LIN {X 0,Y 418.237,Z 526.484,A -85,B 0,C 180,E1 -10180.896,E2 -10180.896} C_VEL
LIN {X 0,Y 419.028,Z 517.254,A -85,B 0,C 180,E1 -10182.347,E2 -10182.347} C_VEL
LIN {X 0,Y 419.709,Z 507.688,A -85,B 0,C 180,E1 -10183.557,E2 -10183.557} C_VEL
LIN {X 0,Y 420.529,Z 497.102,A -85,B 0,C 180,E1 -10184.641,E2 -10184.641} C_VEL
LIN {X 0,Y 421.367,Z 485.277,A -85,B 0,C 180,E1 -10185.601,E2 -10185.601} C_VEL
LIN {X 0,Y 422.297,Z 472.62,A -85,B 0,C 180,E1 -10186.372,E2 -10186.372} C_VEL
LIN {X 0,Y 422.924,Z 459.994,A -85,B 0,C 180,E1 -10186.937,E2 -10186.937} C_VEL
LIN {X 0,Y 423.479,Z 446.573,A -85,B 0,C 180,E1 -10187.318,E2 -10187.318} C_VEL
LIN {X 0,Y 424.411,Z 367.767,A -85,B 0,C 180,E1 -10188.682,E2 -10188.682} C_VEL
LIN {X 0,Y 421.017,Z 346.244,A -85,B 0,C 180,E1 -10189.244,E2 -10189.244} C_VEL
LIN {X 0,Y 419.876,Z 339.849,A -85,B 0,C 180,E1 -10189.436,E2 -10189.436} C_VEL
LIN {X 0,Y 421.122,Z 320.957,A -85,B 0,C 180,E1 -10193,E2 -10193} C_VEL
LIN {X 0,Y 421.806,Z 311.137,A -85,B 0,C 180,E1 -10194.879,E2 -10194.879} C_VEL
LIN {X 0,Y 420.145,Z 301.746,A -85,B 0,C 180,E1 -10196.849,E2 -10196.849} C_VEL
LIN {X 0,Y 418.293,Z 293.389,A -85,B 0,C 180,E1 -10198.701,E2 -10198.701} C_VEL
LIN {X 0,Y 418.243,Z 293.391,A -85,B 0,C 180,E1 -10202.528,E2 -10202.528} C_VEL
LIN {X 0,Y 418.256,Z 293.389,A -85,B 0,C 180,E1 -10204.841,E2 -10204.841} C_VEL
LIN {X 0,Y 418.242,Z 293.39,A -85,B 0,C 180,E1 -10208.442,E2 -10208.442} C_VEL
LIN {X 0,Y 418.219,Z 293.387,A -85,B 0,C 180,E1 -10210.947,E2 -10210.947} C_VEL
LIN {X 0,Y 418.207,Z 293.389,A -85,B 0,C 180,E1 -10213.729,E2 -10213.729} C_VEL
LIN {X 0,Y 418.206,Z 293.391,A -85,B 0,C 180,E1 -10216.448,E2 -10216.448} C_VEL
LIN {X 0,Y 418.221,Z 293.385,A -85,B 0,C 180,E1 -10219.13,E2 -10219.13} C_VEL
LIN {X 0,Y 418.226,Z 293.386,A -85,B 0,C 180,E1 -10222.166,E2 -10222.166} C_VEL
LIN {X 0,Y 418.26,Z 293.378,A -85,B 0,C 180,E1 -10225.42,E2 -10225.42} C_VEL
LIN {X 0,Y 418.208,Z 293.388,A -85,B 0,C 180,E1 -10228.604,E2 -10228.604} C_VEL
LIN {X 0,Y 418.287,Z 293.375,A -85,B 0,C 180,E1 -10231.936,E2 -10231.936} C_VEL
LIN {X 0,Y 418.286,Z 293.375,A -85,B 0,C 180,E1 -10235.163,E2 -10235.163} C_VEL
LIN {X 0,Y 418.231,Z 293.387,A -85,B 0,C 180,E1 -10238.304,E2 -10238.304} C_VEL
LIN {X 0,Y 418.281,Z 293.38,A -85,B 0,C 180,E1 -10241.383,E2 -10241.383} C_VEL
LIN {X 0,Y 418.299,Z 293.375,A -85,B 0,C 180,E1 -10244.406,E2 -10244.406} C_VEL
LIN {X 0,Y 418.352,Z 293.366,A -85,B 0,C 180,E1 -10247.386,E2 -10247.386} C_VEL
LIN {X 0,Y 418.338,Z 293.374,A -85,B 0,C 180,E1 -10250.329,E2 -10250.329} C_VEL
LIN {X 0,Y 418.509,Z 293.347,A -85,B 0,C 180,E1 -10252.28,E2 -10252.28} C_VEL
LIN {X 0,Y 418.51,Z 293.351,A -85,B 0,C 180,E1 -10254.217,E2 -10254.217} C_VEL
LIN {X 0,Y 418.542,Z 293.346,A -85,B 0,C 180,E1 -10258.076,E2 -10258.076} C_VEL
LIN {X 0,Y 418.67,Z 293.327,A -85,B 0,C 180,E1 -10260,E2 -10260} C_VEL
LIN {X 0,Y 418.507,Z 293.356,A -85,B 0,C 180,E1 -10262.888,E2 -10262.888} C_VEL
LIN {X 0,Y 418.491,Z 293.355,A -85,B 0,C 180,E1 -10266.751,E2 -10266.751} C_VEL
LIN {X 0,Y 418.397,Z 293.366,A -85,B 0,C 180,E1 -10268.695,E2 -10268.695} C_VEL
LIN {X 0,Y 418.313,Z 293.375,A -85,B 0,C 180,E1 -10271.631,E2 -10271.631} C_VEL
LIN {X 0,Y 418.3,Z 293.376,A -85,B 0,C 180,E1 -10274.597,E2 -10274.597} C_VEL
LIN {X 0,Y 418.283,Z 293.378,A -85,B 0,C 180,E1 -10277.604,E2 -10277.604} C_VEL
LIN {X 0,Y 418.247,Z 293.385,A -85,B 0,C 180,E1 -10280.664,E2 -10280.664} C_VEL
LIN {X 0,Y 418.283,Z 293.379,A -85,B 0,C 180,E1 -10283.782,E2 -10283.782} C_VEL
LIN {X 0,Y 418.308,Z 293.38,A -85,B 0,C 180,E1 -10287.071,E2 -10287.071} C_VEL
LIN {X 0,Y 418.242,Z 293.383,A -85,B 0,C 180,E1 -10290.273,E2 -10290.273} C_VEL
LIN {X 0,Y 418.246,Z 293.385,A -85,B 0,C 180,E1 -10293.678,E2 -10293.678} C_VEL
LIN {X 0,Y 418.237,Z 293.389,A -85,B 0,C 180,E1 -10297.225,E2 -10297.225} C_VEL
LIN {X 0,Y 418.227,Z 293.388,A -85,B 0,C 180,E1 -10299.685,E2 -10299.685} C_VEL
LIN {X 0,Y 418.213,Z 293.388,A -85,B 0,C 180,E1 -10302.32,E2 -10302.32} C_VEL
LIN {X 0,Y 418.235,Z 293.39,A -85,B 0,C 180,E1 -10305.109,E2 -10305.109} C_VEL
LIN {X 0,Y 418.222,Z 293.39,A -85,B 0,C 180,E1 -10307.765,E2 -10307.765} C_VEL
LIN {X 0,Y 418.235,Z 293.39,A -85,B 0,C 180,E1 -10311.557,E2 -10311.557} C_VEL
LIN {X 0,Y 418.258,Z 293.381,A -85,B 0,C 180,E1 -10315.16,E2 -10315.16} C_VEL
LIN {X 0,Y 418.246,Z 293.386,A -85,B 0,C 180,E1 -10317.473,E2 -10317.473} C_VEL
LIN {X 0,Y 418.265,Z 293.452,A -85,B 0,C 180,E1 -10319.201,E2 -10319.201} C_VEL
LIN {X 0,Y 420.275,Z 303.434,A -85,B 0,C 180,E1 -10321.525,E2 -10321.525} C_VEL
LIN {X 0,Y 420.363,Z 304.121,A -85,B 0,C 180,E1 -10321.647,E2 -10321.647} C_VEL
LIN {X 0,Y 424.619,Z 321.891,A -85,B 0,C 180,E1 -10322.199,E2 -10322.199} C_VEL
LIN {X 0,Y 424.878,Z 325.308,A -85,B 0,C 180,E1 -10322.274,E2 -10322.274} C_VEL
LIN {X 0,Y 423.654,Z 411.995,A -85,B 0,C 180,E1 -10323.783,E2 -10323.783} C_VEL
LIN {X 0,Y 423.327,Z 425.918,A -85,B 0,C 180,E1 -10324.246,E2 -10324.246} C_VEL
LIN {X 0,Y 422.698,Z 438.277,A -85,B 0,C 180,E1 -10324.849,E2 -10324.849} C_VEL
LIN {X 0,Y 422.001,Z 450.37,A -85,B 0,C 180,E1 -10325.658,E2 -10325.658} C_VEL
LIN {X 0,Y 421.34,Z 460.803,A -85,B 0,C 180,E1 -10326.551,E2 -10326.551} C_VEL
LIN {X 0,Y 420.519,Z 471.216,A -85,B 0,C 180,E1 -10327.654,E2 -10327.654} C_VEL
LIN {X 0,Y 419.787,Z 480.656,A -85,B 0,C 180,E1 -10328.904,E2 -10328.904} C_VEL
LIN {X 0,Y 418.974,Z 489.748,A -85,B 0,C 180,E1 -10330.399,E2 -10330.399} C_VEL
LIN {X 0,Y 418.366,Z 497.004,A -85,B 0,C 180,E1 -10331.895,E2 -10331.895} C_VEL
LIN {X 0,Y 417.912,Z 502.928,A -85,B 0,C 180,E1 -10333.451,E2 -10333.451} C_VEL
LIN {X 0,Y 417.571,Z 507.193,A -85,B 0,C 180,E1 -10334.879,E2 -10334.879} C_VEL
LIN {X 0,Y 417.319,Z 510.544,A -85,B 0,C 180,E1 -10336.364,E2 -10336.364} C_VEL
LIN {X 0,Y 417.186,Z 512.718,A -85,B 0,C 180,E1 -10337.712,E2 -10337.712} C_VEL
LIN {X 0,Y 417.034,Z 514.334,A -85,B 0,C 180,E1 -10339.52,E2 -10339.52} C_VEL
LIN {X 0,Y 417.041,Z 514.637,A -85,B 0,C 180,E1 -10341.277,E2 -10341.277} C_VEL
LIN {X 0,Y 417.072,Z 514.25,A -85,B 0,C 180,E1 -10342.253,E2 -10342.253} C_VEL
LIN {X 0,Y 417.181,Z 512.868,A -85,B 0,C 180,E1 -10343.724,E2 -10343.724} C_VEL
LIN {X 0,Y 416.533,Z 511.788,A -85,B 0,C 180,E1 -10344.516,E2 -10344.516} C_VEL
LIN {X 0,Y 413.788,Z 509.541,A -85,B 0,C 180,E1 -10345.795,E2 -10345.795} C_VEL
LIN {X 0,Y 411.494,Z 507.287,A -85,B 0,C 180,E1 -10346.808,E2 -10346.808} C_VEL
LIN {X 0,Y 410.54,Z 505.221,A -85,B 0,C 180,E1 -10347.572,E2 -10347.572} C_VEL
LIN {X 0,Y 410.478,Z 504.425,A -85,B 0,C 180,E1 -10347.826,E2 -10347.826} C_VEL
LIN {X 0,Y 410.657,Z 500.332,A -85,B 0,C 180,E1 -10349.02,E2 -10349.02} C_VEL
LIN {X 0,Y 411.218,Z 494.07,A -85,B 0,C 180,E1 -10350.49,E2 -10350.49} C_VEL
LIN {X 0,Y 411.727,Z 486.262,A -85,B 0,C 180,E1 -10351.957,E2 -10351.957} C_VEL
LIN {X 0,Y 412.392,Z 476.551,A -85,B 0,C 180,E1 -10353.42,E2 -10353.42} C_VEL
LIN {X 0,Y 413.042,Z 466.441,A -85,B 0,C 180,E1 -10354.636,E2 -10354.636} C_VEL
LIN {X 0,Y 413.78,Z 455.013,A -85,B 0,C 180,E1 -10355.727,E2 -10355.727} C_VEL
LIN {X 0,Y 414.492,Z 443.752,A -85,B 0,C 180,E1 -10356.573,E2 -10356.573} C_VEL
LIN {X 0,Y 414.845,Z 432.31,A -85,B 0,C 180,E1 -10357.239,E2 -10357.239} C_VEL
LIN {X 0,Y 415.282,Z 419.113,A -85,B 0,C 180,E1 -10357.782,E2 -10357.782} C_VEL
LIN {X 0,Y 415.62,Z 406.202,A -85,B 0,C 180,E1 -10358.112,E2 -10358.112} C_VEL
LIN {X 0,Y 416.569,Z 323.375,A -85,B 0,C 180,E1 -10359.537,E2 -10359.537} C_VEL
LIN {X 0,Y 412.825,Z 304.032,A -85,B 0,C 180,E1 -10360.041,E2 -10360.041} C_VEL
LIN {X 0,Y 411.358,Z 294.341,A -85,B 0,C 180,E1 -10362.238,E2 -10362.238} C_VEL
LIN {X 0,Y 411.258,Z 294.253,A -85,B 0,C 180,E1 -10365.869,E2 -10365.869} C_VEL
LIN {X 0,Y 411.224,Z 294.262,A -85,B 0,C 180,E1 -10368.949,E2 -10368.949} C_VEL
LIN {X 0,Y 411.205,Z 294.264,A -85,B 0,C 180,E1 -10372.641,E2 -10372.641} C_VEL
LIN {X 0,Y 411.189,Z 294.264,A -85,B 0,C 180,E1 -10375.297,E2 -10375.297} C_VEL
LIN {X 0,Y 411.177,Z 294.266,A -85,B 0,C 180,E1 -10378.594,E2 -10378.594} C_VEL
LIN {X 0,Y 411.168,Z 294.263,A -85,B 0,C 180,E1 -10381.998,E2 -10381.998} C_VEL
LIN {X 0,Y 411.208,Z 294.264,A -85,B 0,C 180,E1 -10384.877,E2 -10384.877} C_VEL
LIN {X 0,Y 411.2,Z 294.259,A -85,B 0,C 180,E1 -10388.167,E2 -10388.167} C_VEL
LIN {X 0,Y 411.165,Z 294.265,A -85,B 0,C 180,E1 -10391.808,E2 -10391.808} C_VEL
LIN {X 0,Y 411.179,Z 294.267,A -85,B 0,C 180,E1 -10395.509,E2 -10395.509} C_VEL
LIN {X 0,Y 411.152,Z 294.267,A -85,B 0,C 180,E1 -10398.775,E2 -10398.775} C_VEL
LIN {X 0,Y 411.188,Z 294.263,A -85,B 0,C 180,E1 -10402.025,E2 -10402.025} C_VEL
LIN {X 0,Y 411.207,Z 294.261,A -85,B 0,C 180,E1 -10405.123,E2 -10405.123} C_VEL
LIN {X 0,Y 411.169,Z 294.266,A -85,B 0,C 180,E1 -10408.003,E2 -10408.003} C_VEL
LIN {X 0,Y 411.198,Z 294.264,A -85,B 0,C 180,E1 -10411.408,E2 -10411.408} C_VEL
LIN {X 0,Y 411.217,Z 294.258,A -85,B 0,C 180,E1 -10414.934,E2 -10414.934} C_VEL
LIN {X 0,Y 411.208,Z 294.265,A -85,B 0,C 180,E1 -10417.913,E2 -10417.913} C_VEL
LIN {X 0,Y 411.223,Z 294.257,A -85,B 0,C 180,E1 -10421.051,E2 -10421.051} C_VEL
LIN {X 0,Y 411.258,Z 294.258,A -85,B 0,C 180,E1 -10424.131,E2 -10424.131} C_VEL
LIN {X 0,Y 411.307,Z 294.246,A -85,B 0,C 180,E1 -10427.165,E2 -10427.165} C_VEL
LIN {X 0,Y 411.282,Z 294.256,A -85,B 0,C 180,E1 -10430.161,E2 -10430.161} C_VEL
LIN {X 0,Y 411.395,Z 294.235,A -85,B 0,C 180,E1 -10433.132,E2 -10433.132} C_VEL
LIN {X 0,Y 411.293,Z 294.248,A -85,B 0,C 180,E1 -10435.099,E2 -10435.099} C_VEL
LIN {X 0,Y 411.506,Z 294.226,A -85,B 0,C 180,E1 -10438.042,E2 -10438.042} C_VEL
LIN {X 0,Y 411.421,Z 294.233,A -85,B 0,C 180,E1 -10440.979,E2 -10440.979} C_VEL
LIN {X 0,Y 411.43,Z 294.232,A -85,B 0,C 180,E1 -10442.937,E2 -10442.937} C_VEL
LIN {X 0,Y 411.394,Z 294.238,A -85,B 0,C 180,E1 -10446.868,E2 -10446.868} C_VEL
LIN {X 0,Y 411.278,Z 294.251,A -85,B 0,C 180,E1 -10449.839,E2 -10449.839} C_VEL
LIN {X 0,Y 411.309,Z 294.248,A -85,B 0,C 180,E1 -10453.103,E2 -10453.103} C_VEL
LIN {X 0,Y 411.261,Z 294.257,A -85,B 0,C 180,E1 -10456.888,E2 -10456.888} C_VEL
LIN {X 0,Y 411.235,Z 294.256,A -85,B 0,C 180,E1 -10459.986,E2 -10459.986} C_VEL
LIN {X 0,Y 411.191,Z 294.264,A -85,B 0,C 180,E1 -10463.148,E2 -10463.148} C_VEL
LIN {X 0,Y 411.178,Z 294.264,A -85,B 0,C 180,E1 -10466.385,E2 -10466.385} C_VEL
LIN {X 0,Y 411.198,Z 294.26,A -85,B 0,C 180,E1 -10469.713,E2 -10469.713} C_VEL
LIN {X 0,Y 411.207,Z 294.265,A -85,B 0,C 180,E1 -10473.156,E2 -10473.156} C_VEL
LIN {X 0,Y 411.195,Z 294.262,A -85,B 0,C 180,E1 -10476.552,E2 -10476.552} C_VEL
LIN {X 0,Y 411.172,Z 294.264,A -85,B 0,C 180,E1 -10479.72,E2 -10479.72} C_VEL
LIN {X 0,Y 411.165,Z 294.27,A -85,B 0,C 180,E1 -10483.135,E2 -10483.135} C_VEL
LIN {X 0,Y 411.166,Z 294.265,A -85,B 0,C 180,E1 -10485.881,E2 -10485.881} C_VEL
LIN {X 0,Y 411.16,Z 294.271,A -85,B 0,C 180,E1 -10489.492,E2 -10489.492} C_VEL
LIN {X 0,Y 411.185,Z 294.263,A -85,B 0,C 180,E1 -10492.025,E2 -10492.025} C_VEL
LIN {X 0,Y 411.205,Z 294.262,A -85,B 0,C 180,E1 -10495.123,E2 -10495.123} C_VEL
LIN {X 0,Y 411.167,Z 294.27,A -85,B 0,C 180,E1 -10498.002,E2 -10498.002} C_VEL
LIN {X 0,Y 411.214,Z 294.264,A -85,B 0,C 180,E1 -10501.409,E2 -10501.409} C_VEL
LIN {X 0,Y 411.262,Z 294.307,A -85,B 0,C 180,E1 -10502.073,E2 -10502.073} C_VEL
LIN {X 0,Y 413.901,Z 307.893,A -85,B 0,C 180,E1 -10504.88,E2 -10504.88} C_VEL
LIN {X 0,Y 414.052,Z 312.05,A -85,B 0,C 180,E1 -10505.693,E2 -10505.693} C_VEL
LIN {X 0,Y 412.954,Z 329.844,A -85,B 0,C 180,E1 -10509.059,E2 -10509.059} C_VEL
LIN {X 0,Y 412.351,Z 339.884,A -85,B 0,C 180,E1 -10510.943,E2 -10510.943} C_VEL
LIN {X 0,Y 416.255,Z 368.768,A -85,B 0,C 180,E1 -10511.625,E2 -10511.625} C_VEL
LIN {X 0,Y 415.383,Z 449.072,A -85,B 0,C 180,E1 -10513.03,E2 -10513.03} C_VEL
LIN {X 0,Y 414.775,Z 463.016,A -85,B 0,C 180,E1 -10513.48,E2 -10513.48} C_VEL
LIN {X 0,Y 414.176,Z 476.032,A -85,B 0,C 180,E1 -10514.12,E2 -10514.12} C_VEL
LIN {X 0,Y 413.358,Z 488.654,A -85,B 0,C 180,E1 -10514.972,E2 -10514.972} C_VEL
LIN {X 0,Y 412.697,Z 500.406,A -85,B 0,C 180,E1 -10516.003,E2 -10516.003} C_VEL
LIN {X 0,Y 411.956,Z 511.029,A -85,B 0,C 180,E1 -10517.186,E2 -10517.186} C_VEL
LIN {X 0,Y 411.342,Z 520.018,A -85,B 0,C 180,E1 -10518.418,E2 -10518.418} C_VEL
LIN {X 0,Y 410.749,Z 528.786,A -85,B 0,C 180,E1 -10519.899,E2 -10519.899} C_VEL
LIN {X 0,Y 410.387,Z 535.776,A -85,B 0,C 180,E1 -10521.381,E2 -10521.381} C_VEL
LIN {X 0,Y 410.162,Z 542.192,A -85,B 0,C 180,E1 -10523.111,E2 -10523.111} C_VEL
LIN {X 0,Y 410.032,Z 546.387,A -85,B 0,C 180,E1 -10524.59,E2 -10524.59} C_VEL
LIN {X 0,Y 409.943,Z 549.506,A -85,B 0,C 180,E1 -10526.067,E2 -10526.067} C_VEL
LIN {X 0,Y 409.987,Z 551.061,A -85,B 0,C 180,E1 -10527.052,E2 -10527.052} C_VEL
LIN {X 0,Y 410.019,Z 552.161,A -85,B 0,C 180,E1 -10528.035,E2 -10528.035} C_VEL
LIN {X 0,Y 409.973,Z 553.147,A -85,B 0,C 180,E1 -10529.999,E2 -10529.999} C_VEL
LIN {X 0,Y 409.978,Z 553.06,A -85,B 0,C 180,E1 -10530.982,E2 -10530.982} C_VEL
LIN {X 0,Y 410.018,Z 552.548,A -85,B 0,C 180,E1 -10531.964,E2 -10531.964} C_VEL
LIN {X 0,Y 409.969,Z 551.622,A -85,B 0,C 180,E1 -10532.947,E2 -10532.947} C_VEL
LIN {X 0,Y 410.02,Z 548.582,A -85,B 0,C 180,E1 -10534.916,E2 -10534.916} C_VEL
LIN {X 0,Y 410.041,Z 545.565,A -85,B 0,C 180,E1 -10536.223,E2 -10536.223} C_VEL
LIN {X 0,Y 410.283,Z 540.602,A -85,B 0,C 180,E1 -10537.876,E2 -10537.876} C_VEL
LIN {X 0,Y 410.702,Z 533.771,A -85,B 0,C 180,E1 -10539.604,E2 -10539.604} C_VEL
LIN {X 0,Y 411.253,Z 526.369,A -85,B 0,C 180,E1 -10541.084,E2 -10541.084} C_VEL
LIN {X 0,Y 412.072,Z 517.205,A -85,B 0,C 180,E1 -10542.559,E2 -10542.559} C_VEL
LIN {X 0,Y 412.81,Z 507.705,A -85,B 0,C 180,E1 -10543.788,E2 -10543.788} C_VEL
LIN {X 0,Y 413.65,Z 497.196,A -85,B 0,C 180,E1 -10544.89,E2 -10544.89} C_VEL
LIN {X 0,Y 414.555,Z 485.515,A -85,B 0,C 180,E1 -10545.864,E2 -10545.864} C_VEL
LIN {X 0,Y 415.517,Z 473.045,A -85,B 0,C 180,E1 -10546.647,E2 -10546.647} C_VEL
LIN {X 0,Y 416.215,Z 459.929,A -85,B 0,C 180,E1 -10547.25,E2 -10547.25} C_VEL
LIN {X 0,Y 416.778,Z 446.777,A -85,B 0,C 180,E1 -10547.637,E2 -10547.637} C_VEL
LIN {X 0,Y 417.744,Z 368.102,A -85,B 0,C 180,E1 -10549.023,E2 -10549.023} C_VEL
LIN {X 0,Y 414.43,Z 347.438,A -85,B 0,C 180,E1 -10549.58,E2 -10549.58} C_VEL
LIN {X 0,Y 413.028,Z 339.466,A -85,B 0,C 180,E1 -10549.826,E2 -10549.826} C_VEL
LIN {X 0,Y 414.155,Z 323.075,A -85,B 0,C 180,E1 -10552.972,E2 -10552.972} C_VEL
LIN {X 0,Y 414.904,Z 312.386,A -85,B 0,C 180,E1 -10555.053,E2 -10555.053} C_VEL
LIN {X 0,Y 413.209,Z 303.005,A -85,B 0,C 180,E1 -10557.063,E2 -10557.063} C_VEL
LIN {X 0,Y 411.224,Z 294.269,A -85,B 0,C 180,E1 -10559.041,E2 -10559.041} C_VEL
LIN {X 0,Y 411.163,Z 294.27,A -85,B 0,C 180,E1 -10561.997,E2 -10561.997} C_VEL
LIN {X 0,Y 411.207,Z 294.267,A -85,B 0,C 180,E1 -10564.878,E2 -10564.878} C_VEL
LIN {X 0,Y 411.196,Z 294.267,A -85,B 0,C 180,E1 -10568.167,E2 -10568.167} C_VEL
LIN {X 0,Y 411.161,Z 294.265,A -85,B 0,C 180,E1 -10571.228,E2 -10571.228} C_VEL
LIN {X 0,Y 411.173,Z 294.27,A -85,B 0,C 180,E1 -10574.49,E2 -10574.49} C_VEL
LIN {X 0,Y 411.175,Z 294.268,A -85,B 0,C 180,E1 -10578.194,E2 -10578.194} C_VEL
LIN {X 0,Y 411.219,Z 294.261,A -85,B 0,C 180,E1 -10580.776,E2 -10580.776} C_VEL
LIN {X 0,Y 411.194,Z 294.264,A -85,B 0,C 180,E1 -10584.471,E2 -10584.471} C_VEL
LIN {X 0,Y 411.203,Z 294.262,A -85,B 0,C 180,E1 -10586.873,E2 -10586.873} C_VEL
LIN {X 0,Y 411.229,Z 294.261,A -85,B 0,C 180,E1 -10590.644,E2 -10590.644} C_VEL
LIN {X 0,Y 411.233,Z 294.255,A -85,B 0,C 180,E1 -10593.619,E2 -10593.619} C_VEL
LIN {X 0,Y 411.198,Z 294.265,A -85,B 0,C 180,E1 -10596.852,E2 -10596.852} C_VEL
LIN {X 0,Y 411.211,Z 294.254,A -85,B 0,C 180,E1 -10600.05,E2 -10600.05} C_VEL
LIN {X 0,Y 411.259,Z 294.251,A -85,B 0,C 180,E1 -10603.131,E2 -10603.131} C_VEL
LIN {X 0,Y 411.302,Z 294.249,A -85,B 0,C 180,E1 -10606.896,E2 -10606.896} C_VEL
LIN {X 0,Y 411.29,Z 294.251,A -85,B 0,C 180,E1 -10610.161,E2 -10610.161} C_VEL
LIN {X 0,Y 411.478,Z 294.222,A -85,B 0,C 180,E1 -10612.147,E2 -10612.147} C_VEL
LIN {X 0,Y 411.472,Z 294.227,A -85,B 0,C 180,E1 -10614.118,E2 -10614.118} C_VEL
LIN {X 0,Y 411.511,Z 294.221,A -85,B 0,C 180,E1 -10618.043,E2 -10618.043} C_VEL
LIN {X 0,Y 411.639,Z 294.203,A -85,B 0,C 180,E1 -10620,E2 -10620} C_VEL
LIN {X 0,Y 411.462,Z 294.234,A -85,B 0,C 180,E1 -10622.937,E2 -10622.937} C_VEL
LIN {X 0,Y 411.458,Z 294.232,A -85,B 0,C 180,E1 -10626.867,E2 -10626.867} C_VEL
LIN {X 0,Y 411.29,Z 294.247,A -85,B 0,C 180,E1 -10629.839,E2 -10629.839} C_VEL
LIN {X 0,Y 411.302,Z 294.248,A -85,B 0,C 180,E1 -10633.105,E2 -10633.105} C_VEL
LIN {X 0,Y 411.254,Z 294.257,A -85,B 0,C 180,E1 -10636.889,E2 -10636.889} C_VEL
LIN {X 0,Y 411.228,Z 294.257,A -85,B 0,C 180,E1 -10639.987,E2 -10639.987} C_VEL
LIN {X 0,Y 411.2,Z 294.267,A -85,B 0,C 180,E1 -10643.148,E2 -10643.148} C_VEL
LIN {X 0,Y 411.234,Z 294.256,A -85,B 0,C 180,E1 -10646.382,E2 -10646.382} C_VEL
LIN {X 0,Y 411.198,Z 294.263,A -85,B 0,C 180,E1 -10649.713,E2 -10649.713} C_VEL
LIN {X 0,Y 411.205,Z 294.261,A -85,B 0,C 180,E1 -10653.157,E2 -10653.157} C_VEL
LIN {X 0,Y 411.191,Z 294.261,A -85,B 0,C 180,E1 -10656.553,E2 -10656.553} C_VEL
LIN {X 0,Y 411.194,Z 294.264,A -85,B 0,C 180,E1 -10659.725,E2 -10659.725} C_VEL
LIN {X 0,Y 411.164,Z 294.269,A -85,B 0,C 180,E1 -10663.135,E2 -10663.135} C_VEL
LIN {X 0,Y 411.164,Z 294.269,A -85,B 0,C 180,E1 -10665.882,E2 -10665.882} C_VEL
LIN {X 0,Y 411.148,Z 294.27,A -85,B 0,C 180,E1 -10668.775,E2 -10668.775} C_VEL
LIN {X 0,Y 411.183,Z 294.266,A -85,B 0,C 180,E1 -10672.026,E2 -10672.026} C_VEL
LIN {X 0,Y 411.205,Z 294.265,A -85,B 0,C 180,E1 -10675.667,E2 -10675.667} C_VEL
LIN {X 0,Y 411.2,Z 294.319,A -85,B 0,C 180,E1 -10678.878,E2 -10678.878} C_VEL
LIN {X 0,Y 413.33,Z 304.267,A -85,B 0,C 180,E1 -10681.243,E2 -10681.243} C_VEL
LIN {X 0,Y 416.615,Z 316.53,A -85,B 0,C 180,E1 -10681.664,E2 -10681.664} C_VEL
LIN {X 0,Y 418.302,Z 325.142,A -85,B 0,C 180,E1 -10681.915,E2 -10681.915} C_VEL
LIN {X 0,Y 416.98,Z 411.971,A -85,B 0,C 180,E1 -10683.444,E2 -10683.444} C_VEL
LIN {X 0,Y 416.657,Z 425.074,A -85,B 0,C 180,E1 -10683.876,E2 -10683.876} C_VEL
LIN {X 0,Y 416.037,Z 437.678,A -85,B 0,C 180,E1 -10684.485,E2 -10684.485} C_VEL
LIN {X 0,Y 415.362,Z 449.209,A -85,B 0,C 180,E1 -10685.243,E2 -10685.243} C_VEL
LIN {X 0,Y 414.663,Z 459.822,A -85,B 0,C 180,E1 -10686.141,E2 -10686.141} C_VEL
LIN {X 0,Y 413.78,Z 470.539,A -85,B 0,C 180,E1 -10687.27,E2 -10687.27} C_VEL
LIN {X 0,Y 412.969,Z 480.214,A -85,B 0,C 180,E1 -10688.538,E2 -10688.538} C_VEL
LIN {X 0,Y 412.245,Z 487.972,A -85,B 0,C 180,E1 -10689.789,E2 -10689.789} C_VEL
LIN {X 0,Y 411.564,Z 495.689,A -85,B 0,C 180,E1 -10691.327,E2 -10691.327} C_VEL
LIN {X 0,Y 410.948,Z 502.674,A -85,B 0,C 180,E1 -10693.099,E2 -10693.099} C_VEL
LIN {X 0,Y 410.567,Z 507.232,A -85,B 0,C 180,E1 -10694.614,E2 -10694.614} C_VEL
LIN {X 0,Y 410.297,Z 510.665,A -85,B 0,C 180,E1 -10696.126,E2 -10696.126} C_VEL
LIN {X 0,Y 410.13,Z 513.062,A -85,B 0,C 180,E1 -10697.624,E2 -10697.624} C_VEL
LIN {X 0,Y 409.994,Z 514.513,A -85,B 0,C 180,E1 -10699.132,E2 -10699.132} C_VEL
LIN {X 0,Y 409.908,Z 514.954,A -85,B 0,C 180,E1 -10700.128,E2 -10700.128} C_VEL
LIN {X 0,Y 409.976,Z 514.638,A -85,B 0,C 180,E1 -10702.118,E2 -10702.118} C_VEL
LIN {X 0,Y 410.09,Z 513.202,A -85,B 0,C 180,E1 -10703.731,E2 -10703.731} C_VEL
LIN {X 0,Y 410.121,Z 511.149,A -85,B 0,C 180,E1 -10705.085,E2 -10705.085} C_VEL
LIN {X 0,Y 410.328,Z 507.976,A -85,B 0,C 180,E1 -10706.564,E2 -10706.564} C_VEL
LIN {X 0,Y 410.478,Z 504.425,A -85,B 0,C 180,E1 -10707.826,E2 -10707.826} C_VEL
LIN {X 0,Y 409.915,Z 502.016,A -85,B 0,C 180,E1 -10708.576,E2 -10708.576} C_VEL
LIN {X 0,Y 406.247,Z 495.799,A -85,B 0,C 180,E1 -10710.245,E2 -10710.245} C_VEL
LIN {X 0,Y 404.654,Z 491.638,A -85,B 0,C 180,E1 -10711.171,E2 -10711.171} C_VEL
LIN {X 0,Y 404.508,Z 489.298,A -85,B 0,C 180,E1 -10711.622,E2 -10711.622} C_VEL
LIN {X 0,Y 405.101,Z 481.13,A -85,B 0,C 180,E1 -10712.984,E2 -10712.984} C_VEL
LIN {X 0,Y 405.734,Z 472.036,A -85,B 0,C 180,E1 -10714.222,E2 -10714.222} C_VEL
LIN {X 0,Y 406.39,Z 461.925,A -85,B 0,C 180,E1 -10715.334,E2 -10715.334} C_VEL
LIN {X 0,Y 407.183,Z 450.692,A -85,B 0,C 180,E1 -10716.318,E2 -10716.318} C_VEL
LIN {X 0,Y 407.684,Z 440.078,A -85,B 0,C 180,E1 -10717.056,E2 -10717.056} C_VEL
LIN {X 0,Y 408.133,Z 428.554,A -85,B 0,C 180,E1 -10717.67,E2 -10717.67} C_VEL
LIN {X 0,Y 408.508,Z 416.317,A -85,B 0,C 180,E1 -10718.129,E2 -10718.129} C_VEL
LIN {X 0,Y 408.786,Z 400.812,A -85,B 0,C 180,E1 -10718.466,E2 -10718.466} C_VEL
LIN {X 0,Y 409.75,Z 324.356,A -85,B 0,C 180,E1 -10719.799,E2 -10719.799} C_VEL
LIN {X 0,Y 406.056,Z 305.517,A -85,B 0,C 180,E1 -10720.296,E2 -10720.296} C_VEL
LIN {X 0,Y 405.79,Z 304.263,A -85,B 0,C 180,E1 -10720.353,E2 -10720.353} C_VEL
LIN {X 0,Y 404.288,Z 295.127,A -85,B 0,C 180,E1 -10722.487,E2 -10722.487} C_VEL
LIN {X 0,Y 404.226,Z 295.13,A -85,B 0,C 180,E1 -10726.152,E2 -10726.152} C_VEL
LIN {X 0,Y 404.168,Z 295.137,A -85,B 0,C 180,E1 -10729.293,E2 -10729.293} C_VEL
LIN {X 0,Y 404.152,Z 295.145,A -85,B 0,C 180,E1 -10732.831,E2 -10732.831} C_VEL
LIN {X 0,Y 404.142,Z 295.139,A -85,B 0,C 180,E1 -10735.77,E2 -10735.77} C_VEL
LIN {X 0,Y 404.158,Z 295.138,A -85,B 0,C 180,E1 -10739.603,E2 -10739.603} C_VEL
LIN {X 0,Y 404.145,Z 295.141,A -85,B 0,C 180,E1 -10742.622,E2 -10742.622} C_VEL
LIN {X 0,Y 404.181,Z 295.14,A -85,B 0,C 180,E1 -10745.189,E2 -10745.189} C_VEL
LIN {X 0,Y 404.14,Z 295.142,A -85,B 0,C 180,E1 -10748.759,E2 -10748.759} C_VEL
LIN {X 0,Y 404.111,Z 295.146,A -85,B 0,C 180,E1 -10751.597,E2 -10751.597} C_VEL
LIN {X 0,Y 404.149,Z 295.138,A -85,B 0,C 180,E1 -10754.522,E2 -10754.522} C_VEL
LIN {X 0,Y 404.126,Z 295.148,A -85,B 0,C 180,E1 -10757.294,E2 -10757.294} C_VEL
LIN {X 0,Y 404.137,Z 295.141,A -85,B 0,C 180,E1 -10759.951,E2 -10759.951} C_VEL
LIN {X 0,Y 404.137,Z 295.143,A -85,B 0,C 180,E1 -10763.126,E2 -10763.126} C_VEL
LIN {X 0,Y 404.143,Z 295.14,A -85,B 0,C 180,E1 -10766.187,E2 -10766.187} C_VEL
LIN {X 0,Y 404.149,Z 295.145,A -85,B 0,C 180,E1 -10769.715,E2 -10769.715} C_VEL
LIN {X 0,Y 404.134,Z 295.141,A -85,B 0,C 180,E1 -10773.118,E2 -10773.118} C_VEL
LIN {X 0,Y 404.154,Z 295.138,A -85,B 0,C 180,E1 -10776.424,E2 -10776.424} C_VEL
LIN {X 0,Y 404.197,Z 295.14,A -85,B 0,C 180,E1 -10779.874,E2 -10779.874} C_VEL
LIN {X 0,Y 404.221,Z 295.129,A -85,B 0,C 180,E1 -10782.993,E2 -10782.993} C_VEL
LIN {X 0,Y 404.288,Z 295.121,A -85,B 0,C 180,E1 -10786.939,E2 -10786.939} C_VEL
LIN {X 0,Y 404.249,Z 295.132,A -85,B 0,C 180,E1 -10789.988,E2 -10789.988} C_VEL
LIN {X 0,Y 404.345,Z 295.114,A -85,B 0,C 180,E1 -10793.011,E2 -10793.011} C_VEL
LIN {X 0,Y 404.265,Z 295.124,A -85,B 0,C 180,E1 -10795.013,E2 -10795.013} C_VEL
LIN {X 0,Y 404.475,Z 295.102,A -85,B 0,C 180,E1 -10798.008,E2 -10798.008} C_VEL
LIN {X 0,Y 404.388,Z 295.109,A -85,B 0,C 180,E1 -10800.996,E2 -10800.996} C_VEL
LIN {X 0,Y 404.389,Z 295.109,A -85,B 0,C 180,E1 -10802.988,E2 -10802.988} C_VEL
LIN {X 0,Y 404.371,Z 295.113,A -85,B 0,C 180,E1 -10805.985,E2 -10805.985} C_VEL
LIN {X 0,Y 404.258,Z 295.126,A -85,B 0,C 180,E1 -10809.002,E2 -10809.002} C_VEL
LIN {X 0,Y 404.252,Z 295.127,A -85,B 0,C 180,E1 -10812.041,E2 -10812.041} C_VEL
LIN {X 0,Y 404.203,Z 295.133,A -85,B 0,C 180,E1 -10815.118,E2 -10815.118} C_VEL
LIN {X 0,Y 404.207,Z 295.133,A -85,B 0,C 180,E1 -10818.238,E2 -10818.238} C_VEL
LIN {X 0,Y 404.141,Z 295.14,A -85,B 0,C 180,E1 -10821.419,E2 -10821.419} C_VEL
LIN {X 0,Y 404.151,Z 295.143,A -85,B 0,C 180,E1 -10824.667,E2 -10824.667} C_VEL
LIN {X 0,Y 404.106,Z 295.143,A -85,B 0,C 180,E1 -10828.006,E2 -10828.006} C_VEL
LIN {X 0,Y 404.145,Z 295.139,A -85,B 0,C 180,E1 -10830.285,E2 -10830.285} C_VEL
LIN {X 0,Y 404.141,Z 295.139,A -85,B 0,C 180,E1 -10833.813,E2 -10833.813} C_VEL
LIN {X 0,Y 404.138,Z 295.144,A -85,B 0,C 180,E1 -10836.874,E2 -10836.874} C_VEL
LIN {X 0,Y 404.119,Z 295.142,A -85,B 0,C 180,E1 -10840.074,E2 -10840.074} C_VEL
LIN {X 0,Y 404.145,Z 295.144,A -85,B 0,C 180,E1 -10843.082,E2 -10843.082} C_VEL
LIN {X 0,Y 404.123,Z 295.142,A -85,B 0,C 180,E1 -10845.922,E2 -10845.922} C_VEL
LIN {X 0,Y 404.104,Z 295.144,A -85,B 0,C 180,E1 -10848.632,E2 -10848.632} C_VEL
LIN {X 0,Y 404.141,Z 295.146,A -85,B 0,C 180,E1 -10851.495,E2 -10851.495} C_VEL
LIN {X 0,Y 404.176,Z 295.136,A -85,B 0,C 180,E1 -10854.982,E2 -10854.982} C_VEL
LIN {X 0,Y 404.141,Z 295.141,A -85,B 0,C 180,E1 -10858.442,E2 -10858.442} C_VEL
LIN {X 0,Y 404.237,Z 295.241,A -85,B 0,C 180,E1 -10861.862,E2 -10861.862} C_VEL
LIN {X 0,Y 407.043,Z 310.06,A -85,B 0,C 180,E1 -10864.974,E2 -10864.974} C_VEL
LIN {X 0,Y 406.844,Z 316.766,A -85,B 0,C 180,E1 -10866.284,E2 -10866.284} C_VEL
LIN {X 0,Y 405.656,Z 336.078,A -85,B 0,C 180,E1 -10869.99,E2 -10869.99} C_VEL
LIN {X 0,Y 405.398,Z 339.647,A -85,B 0,C 180,E1 -10870.669,E2 -10870.669} C_VEL
LIN {X 0,Y 409.416,Z 369.737,A -85,B 0,C 180,E1 -10871.375,E2 -10871.375} C_VEL
LIN {X 0,Y 408.538,Z 448.32,A -85,B 0,C 180,E1 -10872.769,E2 -10872.769} C_VEL
LIN {X 0,Y 407.946,Z 461.638,A -85,B 0,C 180,E1 -10873.195,E2 -10873.195} C_VEL
LIN {X 0,Y 407.363,Z 473.869,A -85,B 0,C 180,E1 -10873.782,E2 -10873.782} C_VEL
LIN {X 0,Y 406.606,Z 486.191,A -85,B 0,C 180,E1 -10874.588,E2 -10874.588} C_VEL
LIN {X 0,Y 405.85,Z 497.85,A -85,B 0,C 180,E1 -10875.585,E2 -10875.585} C_VEL
LIN {X 0,Y 405.176,Z 508.74,A -85,B 0,C 180,E1 -10876.759,E2 -10876.759} C_VEL
LIN {X 0,Y 404.49,Z 517.772,A -85,B 0,C 180,E1 -10877.965,E2 -10877.965} C_VEL
LIN {X 0,Y 403.773,Z 526.875,A -85,B 0,C 180,E1 -10879.469,E2 -10879.469} C_VEL
LIN {X 0,Y 403.373,Z 534.216,A -85,B 0,C 180,E1 -10880.978,E2 -10880.978} C_VEL
LIN {X 0,Y 403.108,Z 540.083,A -85,B 0,C 180,E1 -10882.486,E2 -10882.486} C_VEL
LIN {X 0,Y 402.967,Z 544.694,A -85,B 0,C 180,E1 -10883.993,E2 -10883.993} C_VEL
LIN {X 0,Y 402.954,Z 547.122,A -85,B 0,C 180,E1 -10884.996,E2 -10884.996} C_VEL
LIN {X 0,Y 402.864,Z 549.104,A -85,B 0,C 180,E1 -10885.998,E2 -10885.998} C_VEL
LIN {X 0,Y 402.887,Z 550.672,A -85,B 0,C 180,E1 -10887,E2 -10887} C_VEL
LIN {X 0,Y 402.948,Z 551.799,A -85,B 0,C 180,E1 -10888,E2 -10888} C_VEL
LIN {X 0,Y 402.896,Z 552.811,A -85,B 0,C 180,E1 -10889.999,E2 -10889.999} C_VEL
LIN {X 0,Y 402.903,Z 552.736,A -85,B 0,C 180,E1 -10890.999,E2 -10890.999} C_VEL
LIN {X 0,Y 402.946,Z 552.249,A -85,B 0,C 180,E1 -10891.998,E2 -10891.998} C_VEL
LIN {X 0,Y 402.859,Z 550.029,A -85,B 0,C 180,E1 -10894.001,E2 -10894.001} C_VEL
LIN {X 0,Y 402.912,Z 547.275,A -85,B 0,C 180,E1 -10895.505,E2 -10895.505} C_VEL
LIN {X 0,Y 403.076,Z 543.507,A -85,B 0,C 180,E1 -10897.01,E2 -10897.01} C_VEL
LIN {X 0,Y 403.325,Z 538.63,A -85,B 0,C 180,E1 -10898.517,E2 -10898.517} C_VEL
LIN {X 0,Y 403.749,Z 532.501,A -85,B 0,C 180,E1 -10900.024,E2 -10900.024} C_VEL
LIN {X 0,Y 404.369,Z 524.904,A -85,B 0,C 180,E1 -10901.529,E2 -10901.529} C_VEL
LIN {X 0,Y 405.126,Z 517.16,A -85,B 0,C 180,E1 -10902.778,E2 -10902.778} C_VEL
LIN {X 0,Y 405.889,Z 507.736,A -85,B 0,C 180,E1 -10904.028,E2 -10904.028} C_VEL
LIN {X 0,Y 406.786,Z 497.307,A -85,B 0,C 180,E1 -10905.147,E2 -10905.147} C_VEL
LIN {X 0,Y 407.754,Z 485.739,A -85,B 0,C 180,E1 -10906.136,E2 -10906.136} C_VEL
LIN {X 0,Y 408.741,Z 473.498,A -85,B 0,C 180,E1 -10906.931,E2 -10906.931} C_VEL
LIN {X 0,Y 409.445,Z 461.417,A -85,B 0,C 180,E1 -10907.512,E2 -10907.512} C_VEL
LIN {X 0,Y 410.03,Z 448.302,A -85,B 0,C 180,E1 -10907.937,E2 -10907.937} C_VEL
LIN {X 0,Y 411.137,Z 369.125,A -85,B 0,C 180,E1 -10909.362,E2 -10909.362} C_VEL
LIN {X 0,Y 407.738,Z 347.833,A -85,B 0,C 180,E1 -10909.95,E2 -10909.95} C_VEL
LIN {X 0,Y 406.165,Z 339.232,A -85,B 0,C 180,E1 -10910.203,E2 -10910.203} C_VEL
LIN {X 0,Y 407.427,Z 321.946,A -85,B 0,C 180,E1 -10913.585,E2 -10913.585} C_VEL
LIN {X 0,Y 407.997,Z 313.64,A -85,B 0,C 180,E1 -10915.234,E2 -10915.234} C_VEL
LIN {X 0,Y 406.237,Z 304.265,A -85,B 0,C 180,E1 -10917.287,E2 -10917.287} C_VEL
LIN {X 0,Y 404.178,Z 295.148,A -85,B 0,C 180,E1 -10919.39,E2 -10919.39} C_VEL
LIN {X 0,Y 404.139,Z 295.149,A -85,B 0,C 180,E1 -10922.621,E2 -10922.621} C_VEL
LIN {X 0,Y 404.178,Z 295.141,A -85,B 0,C 180,E1 -10925.189,E2 -10925.189} C_VEL
LIN {X 0,Y 404.146,Z 295.142,A -85,B 0,C 180,E1 -10928.757,E2 -10928.757} C_VEL
LIN {X 0,Y 404.12,Z 295.142,A -85,B 0,C 180,E1 -10931.599,E2 -10931.599} C_VEL
LIN {X 0,Y 404.142,Z 295.146,A -85,B 0,C 180,E1 -10934.522,E2 -10934.522} C_VEL
LIN {X 0,Y 404.134,Z 295.142,A -85,B 0,C 180,E1 -10937.295,E2 -10937.295} C_VEL
LIN {X 0,Y 404.166,Z 295.137,A -85,B 0,C 180,E1 -10939.955,E2 -10939.955} C_VEL
LIN {X 0,Y 404.133,Z 295.142,A -85,B 0,C 180,E1 -10943.125,E2 -10943.125} C_VEL
LIN {X 0,Y 404.141,Z 295.139,A -85,B 0,C 180,E1 -10946.187,E2 -10946.187} C_VEL
LIN {X 0,Y 404.142,Z 295.138,A -85,B 0,C 180,E1 -10949.715,E2 -10949.715} C_VEL
LIN {X 0,Y 404.191,Z 295.135,A -85,B 0,C 180,E1 -10953.123,E2 -10953.123} C_VEL
LIN {X 0,Y 404.172,Z 295.131,A -85,B 0,C 180,E1 -10955.334,E2 -10955.334} C_VEL
LIN {X 0,Y 404.156,Z 295.142,A -85,B 0,C 180,E1 -10958.582,E2 -10958.582} C_VEL
LIN {X 0,Y 404.207,Z 295.132,A -85,B 0,C 180,E1 -10961.762,E2 -10961.762} C_VEL
LIN {X 0,Y 404.203,Z 295.137,A -85,B 0,C 180,E1 -10964.882,E2 -10964.882} C_VEL
LIN {X 0,Y 404.253,Z 295.121,A -85,B 0,C 180,E1 -10967.959,E2 -10967.959} C_VEL
LIN {X 0,Y 404.43,Z 295.1,A -85,B 0,C 180,E1 -10972.1,E2 -10972.1} C_VEL
LIN {X 0,Y 404.42,Z 295.105,A -85,B 0,C 180,E1 -10974.015,E2 -10974.015} C_VEL
LIN {X 0,Y 404.48,Z 295.097,A -85,B 0,C 180,E1 -10978.009,E2 -10978.009} C_VEL
LIN {X 0,Y 404.608,Z 295.079,A -85,B 0,C 180,E1 -10980,E2 -10980} C_VEL
LIN {X 0,Y 404.419,Z 295.11,A -85,B 0,C 180,E1 -10982.989,E2 -10982.989} C_VEL
LIN {X 0,Y 404.409,Z 295.112,A -85,B 0,C 180,E1 -10986.988,E2 -10986.988} C_VEL
LIN {X 0,Y 404.255,Z 295.123,A -85,B 0,C 180,E1 -10990.012,E2 -10990.012} C_VEL
LIN {X 0,Y 404.263,Z 295.125,A -85,B 0,C 180,E1 -10993.212,E2 -10993.212} C_VEL
LIN {X 0,Y 404.213,Z 295.133,A -85,B 0,C 180,E1 -10997.008,E2 -10997.008} C_VEL
LIN {X 0,Y 404.161,Z 295.138,A -85,B 0,C 180,E1 -11000.352,E2 -11000.352} C_VEL
LIN {X 0,Y 404.166,Z 295.139,A -85,B 0,C 180,E1 -11003.575,E2 -11003.575} C_VEL
LIN {X 0,Y 404.181,Z 295.136,A -85,B 0,C 180,E1 -11005.767,E2 -11005.767} C_VEL
LIN {X 0,Y 404.193,Z 295.133,A -85,B 0,C 180,E1 -11008,E2 -11008} C_VEL
LIN {X 0,Y 404.137,Z 295.14,A -85,B 0,C 180,E1 -11011.559,E2 -11011.559} C_VEL
LIN {X 0,Y 404.182,Z 295.137,A -85,B 0,C 180,E1 -11015.017,E2 -11015.017} C_VEL
LIN {X 0,Y 404.141,Z 295.137,A -85,B 0,C 180,E1 -11018.759,E2 -11018.759} C_VEL
LIN {X 0,Y 404.111,Z 295.148,A -85,B 0,C 180,E1 -11021.599,E2 -11021.599} C_VEL
LIN {X 0,Y 404.143,Z 295.141,A -85,B 0,C 180,E1 -11024.523,E2 -11024.523} C_VEL
LIN {X 0,Y 404.123,Z 295.147,A -85,B 0,C 180,E1 -11027.295,E2 -11027.295} C_VEL
LIN {X 0,Y 404.132,Z 295.145,A -85,B 0,C 180,E1 -11029.952,E2 -11029.952} C_VEL
LIN {X 0,Y 404.132,Z 295.145,A -85,B 0,C 180,E1 -11033.127,E2 -11033.127} C_VEL
LIN {X 0,Y 404.145,Z 295.143,A -85,B 0,C 180,E1 -11036.189,E2 -11036.189} C_VEL
LIN {X 0,Y 404.143,Z 295.255,A -85,B 0,C 180,E1 -11038.555,E2 -11038.555} C_VEL
LIN {X 0,Y 406.2,Z 304.644,A -85,B 0,C 180,E1 -11040.835,E2 -11040.835} C_VEL
LIN {X 0,Y 408.764,Z 312.483,A -85,B 0,C 180,E1 -11041.136,E2 -11041.136} C_VEL
LIN {X 0,Y 411.691,Z 325.22,A -85,B 0,C 180,E1 -11041.543,E2 -11041.543} C_VEL
LIN {X 0,Y 410.331,Z 412.196,A -85,B 0,C 180,E1 -11043.101,E2 -11043.101} C_VEL
LIN {X 0,Y 410.019,Z 425.197,A -85,B 0,C 180,E1 -11043.535,E2 -11043.535} C_VEL
LIN {X 0,Y 409.328,Z 438.224,A -85,B 0,C 180,E1 -11044.172,E2 -11044.172} C_VEL
LIN {X 0,Y 408.617,Z 449.691,A -85,B 0,C 180,E1 -11044.943,E2 -11044.943} C_VEL
LIN {X 0,Y 407.875,Z 460.512,A -85,B 0,C 180,E1 -11045.878,E2 -11045.878} C_VEL
LIN {X 0,Y 406.946,Z 470.967,A -85,B 0,C 180,E1 -11047,E2 -11047} C_VEL
LIN {X 0,Y 406.165,Z 479.729,A -85,B 0,C 180,E1 -11048.16,E2 -11048.16} C_VEL
LIN {X 0,Y 405.437,Z 487.466,A -85,B 0,C 180,E1 -11049.401,E2 -11049.401} C_VEL
LIN {X 0,Y 404.636,Z 495.499,A -85,B 0,C 180,E1 -11050.995,E2 -11050.995} C_VEL
LIN {X 0,Y 403.978,Z 502.596,A -85,B 0,C 180,E1 -11052.798,E2 -11052.798} C_VEL
LIN {X 0,Y 403.581,Z 507.258,A -85,B 0,C 180,E1 -11054.341,E2 -11054.341} C_VEL
LIN {X 0,Y 403.257,Z 510.773,A -85,B 0,C 180,E1 -11055.878,E2 -11055.878} C_VEL
LIN {X 0,Y 403.066,Z 513.414,A -85,B 0,C 180,E1 -11057.54,E2 -11057.54} C_VEL
LIN {X 0,Y 402.941,Z 514.753,A -85,B 0,C 180,E1 -11058.939,E2 -11058.939} C_VEL
LIN {X 0,Y 402.826,Z 515.266,A -85,B 0,C 180,E1 -11059.953,E2 -11059.953} C_VEL
LIN {X 0,Y 402.837,Z 515.339,A -85,B 0,C 180,E1 -11060.967,E2 -11060.967} C_VEL
LIN {X 0,Y 402.952,Z 514.327,A -85,B 0,C 180,E1 -11062.988,E2 -11062.988} C_VEL
LIN {X 0,Y 403.002,Z 513.226,A -85,B 0,C 180,E1 -11063.995,E2 -11063.995} C_VEL
LIN {X 0,Y 403.046,Z 511.684,A -85,B 0,C 180,E1 -11064.999,E2 -11064.999} C_VEL
LIN {X 0,Y 403.239,Z 508.591,A -85,B 0,C 180,E1 -11066.503,E2 -11066.503} C_VEL
LIN {X 0,Y 403.43,Z 504.461,A -85,B 0,C 180,E1 -11068.004,E2 -11068.004} C_VEL
LIN {X 0,Y 403.839,Z 498.165,A -85,B 0,C 180,E1 -11069.751,E2 -11069.751} C_VEL
LIN {X 0,Y 404.378,Z 491.311,A -85,B 0,C 180,E1 -11071.245,E2 -11071.245} C_VEL
LIN {X 0,Y 404.508,Z 489.298,A -85,B 0,C 180,E1 -11071.622,E2 -11071.622} C_VEL
LIN {X 0,Y 404.086,Z 485.689,A -85,B 0,C 180,E1 -11072.282,E2 -11072.282} C_VEL
LIN {X 0,Y 401.665,Z 479.524,A -85,B 0,C 180,E1 -11073.332,E2 -11073.332} C_VEL
LIN {X 0,Y 399.343,Z 472.851,A -85,B 0,C 180,E1 -11074.328,E2 -11074.328} C_VEL
LIN {X 0,Y 399.067,Z 468.371,A -85,B 0,C 180,E1 -11074.886,E2 -11074.886} C_VEL
LIN {X 0,Y 399.788,Z 458.234,A -85,B 0,C 180,E1 -11075.929,E2 -11075.929} C_VEL
LIN {X 0,Y 400.599,Z 445.842,A -85,B 0,C 180,E1 -11076.928,E2 -11076.928} C_VEL
LIN {X 0,Y 401.055,Z 433.733,A -85,B 0,C 180,E1 -11077.679,E2 -11077.679} C_VEL
LIN {X 0,Y 401.544,Z 420.9,A -85,B 0,C 180,E1 -11078.24,E2 -11078.24} C_VEL
LIN {X 0,Y 401.905,Z 408.712,A -85,B 0,C 180,E1 -11078.58,E2 -11078.58} C_VEL
LIN {X 0,Y 402.883,Z 324.925,A -85,B 0,C 180,E1 -11080.078,E2 -11080.078} C_VEL
LIN {X 0,Y 399.372,Z 307.161,A -85,B 0,C 180,E1 -11080.559,E2 -11080.559} C_VEL
LIN {X 0,Y 398.737,Z 304.539,A -85,B 0,C 180,E1 -11080.666,E2 -11080.666} C_VEL
LIN {X 0,Y 397.258,Z 296.001,A -85,B 0,C 180,E1 -11082.696,E2 -11082.696} C_VEL
LIN {X 0,Y 397.172,Z 296.012,A -85,B 0,C 180,E1 -11086.447,E2 -11086.447} C_VEL
LIN {X 0,Y 397.152,Z 296.01,A -85,B 0,C 180,E1 -11089.648,E2 -11089.648} C_VEL
LIN {X 0,Y 397.113,Z 296.019,A -85,B 0,C 180,E1 -11093.031,E2 -11093.031} C_VEL
LIN {X 0,Y 397.082,Z 296.019,A -85,B 0,C 180,E1 -11096.263,E2 -11096.263} C_VEL
LIN {X 0,Y 397.102,Z 296.016,A -85,B 0,C 180,E1 -11099.863,E2 -11099.863} C_VEL
LIN {X 0,Y 397.117,Z 296.019,A -85,B 0,C 180,E1 -11103.273,E2 -11103.273} C_VEL
LIN {X 0,Y 397.111,Z 296.016,A -85,B 0,C 180,E1 -11105.735,E2 -11105.735} C_VEL
LIN {X 0,Y 397.098,Z 296.02,A -85,B 0,C 180,E1 -11108.855,E2 -11108.855} C_VEL
LIN {X 0,Y 397.059,Z 296.021,A -85,B 0,C 180,E1 -11112.269,E2 -11112.269} C_VEL
LIN {X 0,Y 397.09,Z 296.022,A -85,B 0,C 180,E1 -11115.069,E2 -11115.069} C_VEL
LIN {X 0,Y 397.056,Z 296.022,A -85,B 0,C 180,E1 -11118.024,E2 -11118.024} C_VEL
LIN {X 0,Y 397.095,Z 296.021,A -85,B 0,C 180,E1 -11121.724,E2 -11121.724} C_VEL
LIN {X 0,Y 397.122,Z 296.021,A -85,B 0,C 180,E1 -11125.506,E2 -11125.506} C_VEL
LIN {X 0,Y 397.082,Z 296.02,A -85,B 0,C 180,E1 -11129.117,E2 -11129.117} C_VEL
LIN {X 0,Y 397.104,Z 296.016,A -85,B 0,C 180,E1 -11132.603,E2 -11132.603} C_VEL
LIN {X 0,Y 397.116,Z 296.019,A -85,B 0,C 180,E1 -11135.98,E2 -11135.98} C_VEL
LIN {X 0,Y 397.144,Z 296.016,A -85,B 0,C 180,E1 -11139.705,E2 -11139.705} C_VEL
LIN {X 0,Y 397.187,Z 296.005,A -85,B 0,C 180,E1 -11142.845,E2 -11142.845} C_VEL
LIN {X 0,Y 397.234,Z 296,A -85,B 0,C 180,E1 -11146.703,E2 -11146.703} C_VEL
LIN {X 0,Y 397.21,Z 296.007,A -85,B 0,C 180,E1 -11149.808,E2 -11149.808} C_VEL
LIN {X 0,Y 397.298,Z 295.992,A -85,B 0,C 180,E1 -11152.887,E2 -11152.887} C_VEL
LIN {X 0,Y 397.236,Z 295.999,A -85,B 0,C 180,E1 -11154.925,E2 -11154.925} C_VEL
LIN {X 0,Y 397.444,Z 295.977,A -85,B 0,C 180,E1 -11157.973,E2 -11157.973} C_VEL
LIN {X 0,Y 397.443,Z 295.977,A -85,B 0,C 180,E1 -11162.027,E2 -11162.027} C_VEL
LIN {X 0,Y 397.324,Z 295.992,A -85,B 0,C 180,E1 -11166.092,E2 -11166.092} C_VEL
LIN {X 0,Y 397.23,Z 296.001,A -85,B 0,C 180,E1 -11169.162,E2 -11169.162} C_VEL
LIN {X 0,Y 397.217,Z 296.005,A -85,B 0,C 180,E1 -11172.258,E2 -11172.258} C_VEL
LIN {X 0,Y 397.177,Z 296.007,A -85,B 0,C 180,E1 -11175.392,E2 -11175.392} C_VEL
LIN {X 0,Y 397.161,Z 296.014,A -85,B 0,C 180,E1 -11178.573,E2 -11178.573} C_VEL
LIN {X 0,Y 397.098,Z 296.016,A -85,B 0,C 180,E1 -11181.818,E2 -11181.818} C_VEL
LIN {X 0,Y 397.1,Z 296.02,A -85,B 0,C 180,E1 -11185.135,E2 -11185.135} C_VEL
LIN {X 0,Y 397.065,Z 296.023,A -85,B 0,C 180,E1 -11188.548,E2 -11188.548} C_VEL
LIN {X 0,Y 397.082,Z 296.018,A -85,B 0,C 180,E1 -11191.835,E2 -11191.835} C_VEL
LIN {X 0,Y 397.12,Z 296.015,A -85,B 0,C 180,E1 -11194.494,E2 -11194.494} C_VEL
LIN {X 0,Y 397.095,Z 296.017,A -85,B 0,C 180,E1 -11198.276,E2 -11198.276} C_VEL
LIN {X 0,Y 397.054,Z 296.022,A -85,B 0,C 180,E1 -11201.976,E2 -11201.976} C_VEL
LIN {X 0,Y 397.088,Z 296.022,A -85,B 0,C 180,E1 -11205.069,E2 -11205.069} C_VEL
LIN {X 0,Y 397.054,Z 296.023,A -85,B 0,C 180,E1 -11208.023,E2 -11208.023} C_VEL
LIN {X 0,Y 397.093,Z 296.021,A -85,B 0,C 180,E1 -11211.723,E2 -11211.723} C_VEL
LIN {X 0,Y 397.12,Z 296.021,A -85,B 0,C 180,E1 -11215.505,E2 -11215.505} C_VEL
LIN {X 0,Y 397.08,Z 296.021,A -85,B 0,C 180,E1 -11219.117,E2 -11219.117} C_VEL
LIN {X 0,Y 397.185,Z 296.099,A -85,B 0,C 180,E1 -11221.628,E2 -11221.628} C_VEL
LIN {X 0,Y 400.03,Z 310.824,A -85,B 0,C 180,E1 -11224.783,E2 -11224.783} C_VEL
LIN {X 0,Y 400.048,Z 315.248,A -85,B 0,C 180,E1 -11225.671,E2 -11225.671} C_VEL
LIN {X 0,Y 398.736,Z 335.493,A -85,B 0,C 180,E1 -11229.628,E2 -11229.628} C_VEL
LIN {X 0,Y 398.446,Z 339.233,A -85,B 0,C 180,E1 -11230.352,E2 -11230.352} C_VEL
LIN {X 0,Y 402.597,Z 370.193,A -85,B 0,C 180,E1 -11231.109,E2 -11231.109} C_VEL
LIN {X 0,Y 401.661,Z 448.653,A -85,B 0,C 180,E1 -11232.53,E2 -11232.53} C_VEL
LIN {X 0,Y 401.016,Z 462.52,A -85,B 0,C 180,E1 -11232.994,E2 -11232.994} C_VEL
LIN {X 0,Y 400.394,Z 474.976,A -85,B 0,C 180,E1 -11233.623,E2 -11233.623} C_VEL
LIN {X 0,Y 399.608,Z 486.895,A -85,B 0,C 180,E1 -11234.442,E2 -11234.442} C_VEL
LIN {X 0,Y 398.851,Z 498.371,A -85,B 0,C 180,E1 -11235.457,E2 -11235.457} C_VEL
LIN {X 0,Y 398.199,Z 508.278,A -85,B 0,C 180,E1 -11236.551,E2 -11236.551} C_VEL
LIN {X 0,Y 397.487,Z 517.156,A -85,B 0,C 180,E1 -11237.75,E2 -11237.75} C_VEL
LIN {X 0,Y 396.762,Z 526.312,A -85,B 0,C 180,E1 -11239.28,E2 -11239.28} C_VEL
LIN {X 0,Y 396.329,Z 533.693,A -85,B 0,C 180,E1 -11240.816,E2 -11240.816} C_VEL
LIN {X 0,Y 396.042,Z 539.603,A -85,B 0,C 180,E1 -11242.351,E2 -11242.351} C_VEL
LIN {X 0,Y 395.856,Z 544.929,A -85,B 0,C 180,E1 -11244.156,E2 -11244.156} C_VEL
LIN {X 0,Y 395.787,Z 548.699,A -85,B 0,C 180,E1 -11245.926,E2 -11245.926} C_VEL
LIN {X 0,Y 395.789,Z 550.281,A -85,B 0,C 180,E1 -11246.946,E2 -11246.946} C_VEL
LIN {X 0,Y 395.877,Z 551.436,A -85,B 0,C 180,E1 -11247.965,E2 -11247.965} C_VEL
LIN {X 0,Y 395.821,Z 552.474,A -85,B 0,C 180,E1 -11249.999,E2 -11249.999} C_VEL
LIN {X 0,Y 395.831,Z 552.413,A -85,B 0,C 180,E1 -11251.017,E2 -11251.017} C_VEL
LIN {X 0,Y 395.856,Z 551.95,A -85,B 0,C 180,E1 -11252.034,E2 -11252.034} C_VEL
LIN {X 0,Y 395.781,Z 549.758,A -85,B 0,C 180,E1 -11254.072,E2 -11254.072} C_VEL
LIN {X 0,Y 395.824,Z 546.61,A -85,B 0,C 180,E1 -11255.803,E2 -11255.803} C_VEL
LIN {X 0,Y 396.062,Z 541.832,A -85,B 0,C 180,E1 -11257.647,E2 -11257.647} C_VEL
LIN {X 0,Y 396.464,Z 535.573,A -85,B 0,C 180,E1 -11259.437,E2 -11259.437} C_VEL
LIN {X 0,Y 396.987,Z 528.783,A -85,B 0,C 180,E1 -11260.97,E2 -11260.97} C_VEL
LIN {X 0,Y 397.916,Z 520.375,A -85,B 0,C 180,E1 -11262.495,E2 -11262.495} C_VEL
LIN {X 0,Y 398.728,Z 510.507,A -85,B 0,C 180,E1 -11263.928,E2 -11263.928} C_VEL
LIN {X 0,Y 399.73,Z 500.066,A -85,B 0,C 180,E1 -11265.147,E2 -11265.147} C_VEL
LIN {X 0,Y 400.728,Z 489.125,A -85,B 0,C 180,E1 -11266.165,E2 -11266.165} C_VEL
LIN {X 0,Y 401.727,Z 477.007,A -85,B 0,C 180,E1 -11267.039,E2 -11267.039} C_VEL
LIN {X 0,Y 402.526,Z 465.645,A -85,B 0,C 180,E1 -11267.659,E2 -11267.659} C_VEL
LIN {X 0,Y 403.254,Z 452.938,A -85,B 0,C 180,E1 -11268.151,E2 -11268.151} C_VEL
LIN {X 0,Y 403.61,Z 437.795,A -85,B 0,C 180,E1 -11268.496,E2 -11268.496} C_VEL
LIN {X 0,Y 404.509,Z 369.688,A -85,B 0,C 180,E1 -11269.725,E2 -11269.725} C_VEL
LIN {X 0,Y 401.058,Z 348.141,A -85,B 0,C 180,E1 -11270.336,E2 -11270.336} C_VEL
LIN {X 0,Y 399.319,Z 338.793,A -85,B 0,C 180,E1 -11270.636,E2 -11270.636} C_VEL
LIN {X 0,Y 400.549,Z 322.909,A -85,B 0,C 180,E1 -11273.8,E2 -11273.8} C_VEL
LIN {X 0,Y 401.087,Z 314.901,A -85,B 0,C 180,E1 -11275.422,E2 -11275.422} C_VEL
LIN {X 0,Y 399.107,Z 304.568,A -85,B 0,C 180,E1 -11277.737,E2 -11277.737} C_VEL
LIN {X 0,Y 397.114,Z 296.029,A -85,B 0,C 180,E1 -11279.768,E2 -11279.768} C_VEL
LIN {X 0,Y 397.116,Z 296.025,A -85,B 0,C 180,E1 -11283.717,E2 -11283.717} C_VEL
LIN {X 0,Y 397.089,Z 296.02,A -85,B 0,C 180,E1 -11287.208,E2 -11287.208} C_VEL
LIN {X 0,Y 397.099,Z 296.023,A -85,B 0,C 180,E1 -11290.445,E2 -11290.445} C_VEL
LIN {X 0,Y 397.098,Z 296.019,A -85,B 0,C 180,E1 -11293.648,E2 -11293.648} C_VEL
LIN {X 0,Y 397.099,Z 296.02,A -85,B 0,C 180,E1 -11296.52,E2 -11296.52} C_VEL
LIN {X 0,Y 397.111,Z 296.02,A -85,B 0,C 180,E1 -11300.423,E2 -11300.423} C_VEL
LIN {X 0,Y 397.104,Z 296.02,A -85,B 0,C 180,E1 -11304.265,E2 -11304.265} C_VEL
LIN {X 0,Y 397.111,Z 296.02,A -85,B 0,C 180,E1 -11306.727,E2 -11306.727} C_VEL
LIN {X 0,Y 397.121,Z 296.016,A -85,B 0,C 180,E1 -11310.296,E2 -11310.296} C_VEL
LIN {X 0,Y 397.19,Z 296.006,A -85,B 0,C 180,E1 -11312.61,E2 -11312.61} C_VEL
LIN {X 0,Y 397.128,Z 296.009,A -85,B 0,C 180,E1 -11315.982,E2 -11315.982} C_VEL
LIN {X 0,Y 397.135,Z 296.006,A -85,B 0,C 180,E1 -11319.705,E2 -11319.705} C_VEL
LIN {X 0,Y 397.178,Z 296.008,A -85,B 0,C 180,E1 -11322.845,E2 -11322.845} C_VEL
LIN {X 0,Y 397.223,Z 296.006,A -85,B 0,C 180,E1 -11326.679,E2 -11326.679} C_VEL
LIN {X 0,Y 397.214,Z 296.003,A -85,B 0,C 180,E1 -11329.809,E2 -11329.809} C_VEL
LIN {X 0,Y 397.36,Z 295.986,A -85,B 0,C 180,E1 -11332.888,E2 -11332.888} C_VEL
LIN {X 0,Y 397.252,Z 296.001,A -85,B 0,C 180,E1 -11334.925,E2 -11334.925} C_VEL
LIN {X 0,Y 397.448,Z 295.973,A -85,B 0,C 180,E1 -11337.974,E2 -11337.974} C_VEL
LIN {X 0,Y 397.578,Z 295.955,A -85,B 0,C 180,E1 -11340,E2 -11340} C_VEL
LIN {X 0,Y 397.377,Z 295.987,A -85,B 0,C 180,E1 -11343.042,E2 -11343.042} C_VEL
LIN {X 0,Y 397.361,Z 295.989,A -85,B 0,C 180,E1 -11347.112,E2 -11347.112} C_VEL
LIN {X 0,Y 397.215,Z 296,A -85,B 0,C 180,E1 -11350.191,E2 -11350.191} C_VEL
LIN {X 0,Y 397.223,Z 296.001,A -85,B 0,C 180,E1 -11353.321,E2 -11353.321} C_VEL
LIN {X 0,Y 397.179,Z 296.008,A -85,B 0,C 180,E1 -11357.156,E2 -11357.156} C_VEL
LIN {X 0,Y 397.1,Z 296.02,A -85,B 0,C 180,E1 -11360.731,E2 -11360.731} C_VEL
LIN {X 0,Y 397.13,Z 296.013,A -85,B 0,C 180,E1 -11364.019,E2 -11364.019} C_VEL
LIN {X 0,Y 397.192,Z 296.009,A -85,B 0,C 180,E1 -11367.391,E2 -11367.391} C_VEL
LIN {X 0,Y 397.077,Z 296.023,A -85,B 0,C 180,E1 -11370.883,E2 -11370.883} C_VEL
LIN {X 0,Y 397.123,Z 296.014,A -85,B 0,C 180,E1 -11374.494,E2 -11374.494} C_VEL
LIN {X 0,Y 397.094,Z 296.014,A -85,B 0,C 180,E1 -11378.277,E2 -11378.277} C_VEL
LIN {X 0,Y 397.058,Z 296.024,A -85,B 0,C 180,E1 -11380.913,E2 -11380.913} C_VEL
LIN {X 0,Y 397.097,Z 296.021,A -85,B 0,C 180,E1 -11383.65,E2 -11383.65} C_VEL
LIN {X 0,Y 397.097,Z 296.019,A -85,B 0,C 180,E1 -11386.523,E2 -11386.523} C_VEL
LIN {X 0,Y 397.085,Z 296.021,A -85,B 0,C 180,E1 -11390.42,E2 -11390.42} C_VEL
LIN {X 0,Y 397.095,Z 296.021,A -85,B 0,C 180,E1 -11393.005,E2 -11393.005} C_VEL
LIN {X 0,Y 397.119,Z 296.018,A -85,B 0,C 180,E1 -11396.283,E2 -11396.283} C_VEL
LIN {X 0,Y 397.106,Z 296.184,A -85,B 0,C 180,E1 -11398.216,E2 -11398.216} C_VEL
LIN {X 0,Y 399.097,Z 304.962,A -85,B 0,C 180,E1 -11400.396,E2 -11400.396} C_VEL
LIN {X 0,Y 402.153,Z 313.535,A -85,B 0,C 180,E1 -11400.757,E2 -11400.757} C_VEL
LIN {X 0,Y 405.143,Z 326.849,A -85,B 0,C 180,E1 -11401.191,E2 -11401.191} C_VEL
LIN {X 0,Y 403.711,Z 412.796,A -85,B 0,C 180,E1 -11402.756,E2 -11402.756} C_VEL
LIN {X 0,Y 403.368,Z 425.868,A -85,B 0,C 180,E1 -11403.204,E2 -11403.204} C_VEL
LIN {X 0,Y 402.631,Z 438.796,A -85,B 0,C 180,E1 -11403.849,E2 -11403.849} C_VEL
LIN {X 0,Y 401.885,Z 450.193,A -85,B 0,C 180,E1 -11404.632,E2 -11404.632} C_VEL
LIN {X 0,Y 401.008,Z 462.105,A -85,B 0,C 180,E1 -11405.693,E2 -11405.693} C_VEL
LIN {X 0,Y 400.017,Z 472.491,A -85,B 0,C 180,E1 -11406.852,E2 -11406.852} C_VEL
LIN {X 0,Y 399.235,Z 481.033,A -85,B 0,C 180,E1 -11408.033,E2 -11408.033} C_VEL
LIN {X 0,Y 398.262,Z 490.224,A -85,B 0,C 180,E1 -11409.604,E2 -11409.604} C_VEL
LIN {X 0,Y 397.527,Z 497.583,A -85,B 0,C 180,E1 -11411.178,E2 -11411.178} C_VEL
LIN {X 0,Y 397.021,Z 502.512,A -85,B 0,C 180,E1 -11412.487,E2 -11412.487} C_VEL
LIN {X 0,Y 396.566,Z 507.264,A -85,B 0,C 180,E1 -11414.057,E2 -11414.057} C_VEL
LIN {X 0,Y 396.23,Z 510.862,A -85,B 0,C 180,E1 -11415.623,E2 -11415.623} C_VEL
LIN {X 0,Y 396.007,Z 513.764,A -85,B 0,C 180,E1 -11417.449,E2 -11417.449} C_VEL
LIN {X 0,Y 395.859,Z 514.994,A -85,B 0,C 180,E1 -11418.739,E2 -11418.739} C_VEL
LIN {X 0,Y 395.752,Z 515.557,A -85,B 0,C 180,E1 -11419.771,E2 -11419.771} C_VEL
LIN {X 0,Y 395.754,Z 515.69,A -85,B 0,C 180,E1 -11420.804,E2 -11420.804} C_VEL
LIN {X 0,Y 395.864,Z 514.75,A -85,B 0,C 180,E1 -11422.862,E2 -11422.862} C_VEL
LIN {X 0,Y 395.912,Z 513.704,A -85,B 0,C 180,E1 -11423.887,E2 -11423.887} C_VEL
LIN {X 0,Y 395.972,Z 512.217,A -85,B 0,C 180,E1 -11424.909,E2 -11424.909} C_VEL
LIN {X 0,Y 396.151,Z 509.203,A -85,B 0,C 180,E1 -11426.441,E2 -11426.441} C_VEL
LIN {X 0,Y 396.367,Z 505.154,A -85,B 0,C 180,E1 -11427.968,E2 -11427.968} C_VEL
LIN {X 0,Y 396.757,Z 498.95,A -85,B 0,C 180,E1 -11429.747,E2 -11429.747} C_VEL
LIN {X 0,Y 397.33,Z 492.194,A -85,B 0,C 180,E1 -11431.268,E2 -11431.268} C_VEL
LIN {X 0,Y 397.931,Z 483.801,A -85,B 0,C 180,E1 -11432.785,E2 -11432.785} C_VEL
LIN {X 0,Y 398.58,Z 475.173,A -85,B 0,C 180,E1 -11434.045,E2 -11434.045} C_VEL
LIN {X 0,Y 399.067,Z 468.371,A -85,B 0,C 180,E1 -11434.886,E2 -11434.886} C_VEL
LIN {X 0,Y 398.831,Z 463.78,A -85,B 0,C 180,E1 -11435.418,E2 -11435.418} C_VEL
LIN {X 0,Y 396.659,Z 456.072,A -85,B 0,C 180,E1 -11436.26,E2 -11436.26} C_VEL
LIN {X 0,Y 394.339,Z 447.944,A -85,B 0,C 180,E1 -11437.015,E2 -11437.015} C_VEL
LIN {X 0,Y 393.871,Z 442.689,A -85,B 0,C 180,E1 -11437.406,E2 -11437.406} C_VEL
LIN {X 0,Y 394.338,Z 431.239,A -85,B 0,C 180,E1 -11438.069,E2 -11438.069} C_VEL
LIN {X 0,Y 394.805,Z 418.105,A -85,B 0,C 180,E1 -11438.607,E2 -11438.607} C_VEL
LIN {X 0,Y 395.119,Z 405.221,A -85,B 0,C 180,E1 -11438.922,E2 -11438.922} C_VEL
LIN {X 0,Y 396.107,Z 325.954,A -85,B 0,C 180,E1 -11440.354,E2 -11440.354} C_VEL
LIN {X 0,Y 392.657,Z 308.562,A -85,B 0,C 180,E1 -11440.835,E2 -11440.835} C_VEL
LIN {X 0,Y 391.62,Z 304.874,A -85,B 0,C 180,E1 -11440.98,E2 -11440.98} C_VEL
LIN {X 0,Y 390.23,Z 296.876,A -85,B 0,C 180,E1 -11442.931,E2 -11442.931} C_VEL
LIN {X 0,Y 390.144,Z 296.889,A -85,B 0,C 180,E1 -11446.752,E2 -11446.752} C_VEL
LIN {X 0,Y 390.093,Z 296.893,A -85,B 0,C 180,E1 -11450.47,E2 -11450.47} C_VEL
LIN {X 0,Y 390.067,Z 296.894,A -85,B 0,C 180,E1 -11453.353,E2 -11453.353} C_VEL
LIN {X 0,Y 390.036,Z 296.902,A -85,B 0,C 180,E1 -11456.775,E2 -11456.775} C_VEL
LIN {X 0,Y 390.041,Z 296.896,A -85,B 0,C 180,E1 -11460.3,E2 -11460.3} C_VEL
LIN {X 0,Y 390.074,Z 296.891,A -85,B 0,C 180,E1 -11464.025,E2 -11464.025} C_VEL
LIN {X 0,Y 390.045,Z 296.898,A -85,B 0,C 180,E1 -11467.55,E2 -11467.55} C_VEL
LIN {X 0,Y 390.022,Z 296.901,A -85,B 0,C 180,E1 -11470.815,E2 -11470.815} C_VEL
LIN {X 0,Y 390.049,Z 296.896,A -85,B 0,C 180,E1 -11473.884,E2 -11473.884} C_VEL
LIN {X 0,Y 390.052,Z 296.896,A -85,B 0,C 180,E1 -11476.788,E2 -11476.788} C_VEL
LIN {X 0,Y 390.014,Z 296.904,A -85,B 0,C 180,E1 -11479.555,E2 -11479.555} C_VEL
LIN {X 0,Y 390.043,Z 296.895,A -85,B 0,C 180,E1 -11482.45,E2 -11482.45} C_VEL
LIN {X 0,Y 390.066,Z 296.894,A -85,B 0,C 180,E1 -11486.044,E2 -11486.044} C_VEL
LIN {X 0,Y 390.049,Z 296.899,A -85,B 0,C 180,E1 -11489.87,E2 -11489.87} C_VEL
LIN {X 0,Y 390.056,Z 296.896,A -85,B 0,C 180,E1 -11493.227,E2 -11493.227} C_VEL
LIN {X 0,Y 390.071,Z 296.892,A -85,B 0,C 180,E1 -11496.764,E2 -11496.764} C_VEL
LIN {X 0,Y 390.109,Z 296.893,A -85,B 0,C 180,E1 -11499.983,E2 -11499.983} C_VEL
LIN {X 0,Y 390.143,Z 296.883,A -85,B 0,C 180,E1 -11503.248,E2 -11503.248} C_VEL
LIN {X 0,Y 390.2,Z 296.877,A -85,B 0,C 180,E1 -11506.561,E2 -11506.561} C_VEL
LIN {X 0,Y 390.191,Z 296.878,A -85,B 0,C 180,E1 -11510.671,E2 -11510.671} C_VEL
LIN {X 0,Y 390.287,Z 296.868,A -85,B 0,C 180,E1 -11513.797,E2 -11513.797} C_VEL
LIN {X 0,Y 390.411,Z 296.853,A -85,B 0,C 180,E1 -11517.936,E2 -11517.936} C_VEL
LIN {X 0,Y 390.41,Z 296.853,A -85,B 0,C 180,E1 -11522.063,E2 -11522.063} C_VEL
LIN {X 0,Y 390.279,Z 296.87,A -85,B 0,C 180,E1 -11526.202,E2 -11526.202} C_VEL
LIN {X 0,Y 390.188,Z 296.877,A -85,B 0,C 180,E1 -11529.329,E2 -11529.329} C_VEL
LIN {X 0,Y 390.199,Z 296.876,A -85,B 0,C 180,E1 -11533.438,E2 -11533.438} C_VEL
LIN {X 0,Y 390.133,Z 296.885,A -85,B 0,C 180,E1 -11537.298,E2 -11537.298} C_VEL
LIN {X 0,Y 390.091,Z 296.893,A -85,B 0,C 180,E1 -11540.47,E2 -11540.47} C_VEL
LIN {X 0,Y 390.065,Z 296.894,A -85,B 0,C 180,E1 -11543.352,E2 -11543.352} C_VEL
LIN {X 0,Y 390.034,Z 296.902,A -85,B 0,C 180,E1 -11546.774,E2 -11546.774} C_VEL
LIN {X 0,Y 390.039,Z 296.897,A -85,B 0,C 180,E1 -11550.3,E2 -11550.3} C_VEL
LIN {X 0,Y 390.072,Z 296.892,A -85,B 0,C 180,E1 -11554.024,E2 -11554.024} C_VEL
LIN {X 0,Y 390.041,Z 296.896,A -85,B 0,C 180,E1 -11557.78,E2 -11557.78} C_VEL
LIN {X 0,Y 390.019,Z 296.901,A -85,B 0,C 180,E1 -11560.814,E2 -11560.814} C_VEL
LIN {X 0,Y 390.047,Z 296.896,A -85,B 0,C 180,E1 -11563.884,E2 -11563.884} C_VEL
LIN {X 0,Y 390.049,Z 296.896,A -85,B 0,C 180,E1 -11566.788,E2 -11566.788} C_VEL
LIN {X 0,Y 390.012,Z 296.904,A -85,B 0,C 180,E1 -11569.554,E2 -11569.554} C_VEL
LIN {X 0,Y 390.041,Z 296.895,A -85,B 0,C 180,E1 -11572.45,E2 -11572.45} C_VEL
LIN {X 0,Y 390.064,Z 296.894,A -85,B 0,C 180,E1 -11576.044,E2 -11576.044} C_VEL
LIN {X 0,Y 390.047,Z 296.901,A -85,B 0,C 180,E1 -11579.869,E2 -11579.869} C_VEL
LIN {X 0,Y 390.127,Z 297.033,A -85,B 0,C 180,E1 -11581.405,E2 -11581.405} C_VEL
LIN {X 0,Y 392.999,Z 311.579,A -85,B 0,C 180,E1 -11584.583,E2 -11584.583} C_VEL
LIN {X 0,Y 393.116,Z 315.74,A -85,B 0,C 180,E1 -11585.439,E2 -11585.439} C_VEL
LIN {X 0,Y 391.787,Z 334.89,A -85,B 0,C 180,E1 -11589.25,E2 -11589.25} C_VEL
LIN {X 0,Y 391.513,Z 338.977,A -85,B 0,C 180,E1 -11590.057,E2 -11590.057} C_VEL
LIN {X 0,Y 395.781,Z 371.529,A -85,B 0,C 180,E1 -11590.852,E2 -11590.852} C_VEL
LIN {X 0,Y 394.841,Z 447.795,A -85,B 0,C 180,E1 -11592.252,E2 -11592.252} C_VEL
LIN {X 0,Y 394.215,Z 461.073,A -85,B 0,C 180,E1 -11592.692,E2 -11592.692} C_VEL
LIN {X 0,Y 393.536,Z 473.851,A -85,B 0,C 180,E1 -11593.33,E2 -11593.33} C_VEL
LIN {X 0,Y 392.742,Z 485.989,A -85,B 0,C 180,E1 -11594.163,E2 -11594.163} C_VEL
LIN {X 0,Y 391.88,Z 497.564,A -85,B 0,C 180,E1 -11595.193,E2 -11595.193} C_VEL
LIN {X 0,Y 391.227,Z 507.84,A -85,B 0,C 180,E1 -11596.341,E2 -11596.341} C_VEL
LIN {X 0,Y 390.486,Z 516.52,A -85,B 0,C 180,E1 -11597.527,E2 -11597.527} C_VEL
LIN {X 0,Y 389.747,Z 525.738,A -85,B 0,C 180,E1 -11599.085,E2 -11599.085} C_VEL
LIN {X 0,Y 389.283,Z 533.163,A -85,B 0,C 180,E1 -11600.648,E2 -11600.648} C_VEL
LIN {X 0,Y 388.975,Z 539.112,A -85,B 0,C 180,E1 -11602.211,E2 -11602.211} C_VEL
LIN {X 0,Y 388.797,Z 543.935,A -85,B 0,C 180,E1 -11603.824,E2 -11603.824} C_VEL
LIN {X 0,Y 388.729,Z 547.353,A -85,B 0,C 180,E1 -11605.333,E2 -11605.333} C_VEL
LIN {X 0,Y 388.692,Z 549.887,A -85,B 0,C 180,E1 -11606.89,E2 -11606.89} C_VEL
LIN {X 0,Y 388.789,Z 551.069,A -85,B 0,C 180,E1 -11607.927,E2 -11607.927} C_VEL
LIN {X 0,Y 388.761,Z 551.799,A -85,B 0,C 180,E1 -11608.963,E2 -11608.963} C_VEL
LIN {X 0,Y 388.76,Z 552.09,A -85,B 0,C 180,E1 -11611.035,E2 -11611.035} C_VEL
LIN {X 0,Y 388.754,Z 551.648,A -85,B 0,C 180,E1 -11612.071,E2 -11612.071} C_VEL
LIN {X 0,Y 388.705,Z 549.49,A -85,B 0,C 180,E1 -11614.147,E2 -11614.147} C_VEL
LIN {X 0,Y 388.773,Z 545.884,A -85,B 0,C 180,E1 -11616.143,E2 -11616.143} C_VEL
LIN {X 0,Y 389.015,Z 541.638,A -85,B 0,C 180,E1 -11617.787,E2 -11617.787} C_VEL
LIN {X 0,Y 389.44,Z 535.419,A -85,B 0,C 180,E1 -11619.609,E2 -11619.609} C_VEL
LIN {X 0,Y 389.999,Z 528.671,A -85,B 0,C 180,E1 -11621.169,E2 -11621.169} C_VEL
LIN {X 0,Y 390.952,Z 520.325,A -85,B 0,C 180,E1 -11622.721,E2 -11622.721} C_VEL
LIN {X 0,Y 391.774,Z 511.054,A -85,B 0,C 180,E1 -11624.11,E2 -11624.11} C_VEL
LIN {X 0,Y 392.856,Z 500.166,A -85,B 0,C 180,E1 -11625.419,E2 -11625.419} C_VEL
LIN {X 0,Y 393.926,Z 489.364,A -85,B 0,C 180,E1 -11626.452,E2 -11626.452} C_VEL
LIN {X 0,Y 394.969,Z 477.409,A -85,B 0,C 180,E1 -11627.34,E2 -11627.34} C_VEL
LIN {X 0,Y 395.777,Z 466.278,A -85,B 0,C 180,E1 -11627.97,E2 -11627.97} C_VEL
LIN {X 0,Y 396.598,Z 453.067,A -85,B 0,C 180,E1 -11628.5,E2 -11628.5} C_VEL
LIN {X 0,Y 396.988,Z 439.809,A -85,B 0,C 180,E1 -11628.822,E2 -11628.822} C_VEL
LIN {X 0,Y 397.854,Z 369.79,A -85,B 0,C 180,E1 -11630.113,E2 -11630.113} C_VEL
LIN {X 0,Y 394.405,Z 348.648,A -85,B 0,C 180,E1 -11630.731,E2 -11630.731} C_VEL
LIN {X 0,Y 392.469,Z 338.5,A -85,B 0,C 180,E1 -11631.056,E2 -11631.056} C_VEL
LIN {X 0,Y 393.97,Z 321.404,A -85,B 0,C 180,E1 -11634.524,E2 -11634.524} C_VEL
LIN {X 0,Y 394.181,Z 316.167,A -85,B 0,C 180,E1 -11635.617,E2 -11635.617} C_VEL
LIN {X 0,Y 391.92,Z 304.705,A -85,B 0,C 180,E1 -11638.247,E2 -11638.247} C_VEL
LIN {X 0,Y 390.042,Z 296.909,A -85,B 0,C 180,E1 -11640.13,E2 -11640.13} C_VEL
LIN {X 0,Y 390.066,Z 296.902,A -85,B 0,C 180,E1 -11644.024,E2 -11644.024} C_VEL
LIN {X 0,Y 390.039,Z 296.899,A -85,B 0,C 180,E1 -11647.55,E2 -11647.55} C_VEL
LIN {X 0,Y 390.054,Z 296.896,A -85,B 0,C 180,E1 -11650.821,E2 -11650.821} C_VEL
LIN {X 0,Y 390.052,Z 296.898,A -85,B 0,C 180,E1 -11653.886,E2 -11653.886} C_VEL
LIN {X 0,Y 390.054,Z 296.898,A -85,B 0,C 180,E1 -11656.789,E2 -11656.789} C_VEL
LIN {X 0,Y 390.054,Z 296.893,A -85,B 0,C 180,E1 -11659.56,E2 -11659.56} C_VEL
LIN {X 0,Y 390.04,Z 296.897,A -85,B 0,C 180,E1 -11662.449,E2 -11662.449} C_VEL
LIN {X 0,Y 390.064,Z 296.891,A -85,B 0,C 180,E1 -11666.045,E2 -11666.045} C_VEL
LIN {X 0,Y 390.043,Z 296.895,A -85,B 0,C 180,E1 -11669.869,E2 -11669.869} C_VEL
LIN {X 0,Y 390.109,Z 296.888,A -85,B 0,C 180,E1 -11673.232,E2 -11673.232} C_VEL
LIN {X 0,Y 390.102,Z 296.89,A -85,B 0,C 180,E1 -11676.75,E2 -11676.75} C_VEL
LIN {X 0,Y 390.1,Z 296.883,A -85,B 0,C 180,E1 -11679.983,E2 -11679.983} C_VEL
LIN {X 0,Y 390.134,Z 296.881,A -85,B 0,C 180,E1 -11683.248,E2 -11683.248} C_VEL
LIN {X 0,Y 390.191,Z 296.883,A -85,B 0,C 180,E1 -11686.562,E2 -11686.562} C_VEL
LIN {X 0,Y 390.201,Z 296.882,A -85,B 0,C 180,E1 -11690.671,E2 -11690.671} C_VEL
LIN {X 0,Y 390.315,Z 296.862,A -85,B 0,C 180,E1 -11692.759,E2 -11692.759} C_VEL
LIN {X 0,Y 390.224,Z 296.878,A -85,B 0,C 180,E1 -11694.834,E2 -11694.834} C_VEL
LIN {X 0,Y 390.417,Z 296.849,A -85,B 0,C 180,E1 -11697.937,E2 -11697.937} C_VEL
LIN {X 0,Y 390.547,Z 296.83,A -85,B 0,C 180,E1 -11700,E2 -11700} C_VEL
LIN {X 0,Y 390.311,Z 296.866,A -85,B 0,C 180,E1 -11703.097,E2 -11703.097} C_VEL
LIN {X 0,Y 390.306,Z 296.862,A -85,B 0,C 180,E1 -11706.642,E2 -11706.642} C_VEL
LIN {X 0,Y 390.202,Z 296.876,A -85,B 0,C 180,E1 -11709.329,E2 -11709.329} C_VEL
LIN {X 0,Y 390.191,Z 296.877,A -85,B 0,C 180,E1 -11713.439,E2 -11713.439} C_VEL
LIN {X 0,Y 390.146,Z 296.883,A -85,B 0,C 180,E1 -11717.308,E2 -11717.308} C_VEL
LIN {X 0,Y 390.085,Z 296.892,A -85,B 0,C 180,E1 -11720.471,E2 -11720.471} C_VEL
LIN {X 0,Y 390.087,Z 296.896,A -85,B 0,C 180,E1 -11723.351,E2 -11723.351} C_VEL
LIN {X 0,Y 390.111,Z 296.889,A -85,B 0,C 180,E1 -11726.769,E2 -11726.769} C_VEL
LIN {X 0,Y 390.037,Z 296.897,A -85,B 0,C 180,E1 -11730.3,E2 -11730.3} C_VEL
LIN {X 0,Y 390.066,Z 296.893,A -85,B 0,C 180,E1 -11734.025,E2 -11734.025} C_VEL
LIN {X 0,Y 390.039,Z 296.897,A -85,B 0,C 180,E1 -11737.551,E2 -11737.551} C_VEL
LIN {X 0,Y 390.029,Z 296.899,A -85,B 0,C 180,E1 -11740.818,E2 -11740.818} C_VEL
LIN {X 0,Y 390.051,Z 296.898,A -85,B 0,C 180,E1 -11743.887,E2 -11743.887} C_VEL
LIN {X 0,Y 390.051,Z 296.898,A -85,B 0,C 180,E1 -11746.79,E2 -11746.79} C_VEL
LIN {X 0,Y 390.009,Z 296.904,A -85,B 0,C 180,E1 -11749.555,E2 -11749.555} C_VEL
LIN {X 0,Y 390.038,Z 296.899,A -85,B 0,C 180,E1 -11752.451,E2 -11752.451} C_VEL
LIN {X 0,Y 390.069,Z 296.898,A -85,B 0,C 180,E1 -11755.976,E2 -11755.976} C_VEL
LIN {X 0,Y 390.077,Z 296.99,A -85,B 0,C 180,E1 -11757.833,E2 -11757.833} C_VEL
LIN {X 0,Y 391.966,Z 305.333,A -85,B 0,C 180,E1 -11759.949,E2 -11759.949} C_VEL
LIN {X 0,Y 395.835,Z 315.561,A -85,B 0,C 180,E1 -11760.401,E2 -11760.401} C_VEL
LIN {X 0,Y 398.603,Z 327.993,A -85,B 0,C 180,E1 -11760.816,E2 -11760.816} C_VEL
LIN {X 0,Y 397.1,Z 413.302,A -85,B 0,C 180,E1 -11762.395,E2 -11762.395} C_VEL
LIN {X 0,Y 396.721,Z 426.57,A -85,B 0,C 180,E1 -11762.861,E2 -11762.861} C_VEL
LIN {X 0,Y 395.95,Z 439.384,A -85,B 0,C 180,E1 -11763.516,E2 -11763.516} C_VEL
LIN {X 0,Y 395.176,Z 450.712,A -85,B 0,C 180,E1 -11764.311,E2 -11764.311} C_VEL
LIN {X 0,Y 394.25,Z 462.573,A -85,B 0,C 180,E1 -11765.388,E2 -11765.388} C_VEL
LIN {X 0,Y 393.206,Z 472.938,A -85,B 0,C 180,E1 -11766.567,E2 -11766.567} C_VEL
LIN {X 0,Y 392.301,Z 482.284,A -85,B 0,C 180,E1 -11767.902,E2 -11767.902} C_VEL
LIN {X 0,Y 391.285,Z 491.318,A -85,B 0,C 180,E1 -11769.498,E2 -11769.498} C_VEL
LIN {X 0,Y 390.511,Z 498.512,A -85,B 0,C 180,E1 -11771.099,E2 -11771.099} C_VEL
LIN {X 0,Y 389.867,Z 504.589,A -85,B 0,C 180,E1 -11772.828,E2 -11772.828} C_VEL
LIN {X 0,Y 389.31,Z 509.872,A -85,B 0,C 180,E1 -11774.826,E2 -11774.826} C_VEL
LIN {X 0,Y 389.004,Z 512.839,A -85,B 0,C 180,E1 -11776.417,E2 -11776.417} C_VEL
LIN {X 0,Y 388.926,Z 514.245,A -85,B 0,C 180,E1 -11777.477,E2 -11777.477} C_VEL
LIN {X 0,Y 388.686,Z 515.835,A -85,B 0,C 180,E1 -11779.583,E2 -11779.583} C_VEL
LIN {X 0,Y 388.664,Z 516.036,A -85,B 0,C 180,E1 -11780.635,E2 -11780.635} C_VEL
LIN {X 0,Y 388.773,Z 515.171,A -85,B 0,C 180,E1 -11782.731,E2 -11782.731} C_VEL
LIN {X 0,Y 388.837,Z 514.161,A -85,B 0,C 180,E1 -11783.775,E2 -11783.775} C_VEL
LIN {X 0,Y 388.877,Z 512.747,A -85,B 0,C 180,E1 -11784.816,E2 -11784.816} C_VEL
LIN {X 0,Y 389.047,Z 509.805,A -85,B 0,C 180,E1 -11786.376,E2 -11786.376} C_VEL
LIN {X 0,Y 389.304,Z 505.833,A -85,B 0,C 180,E1 -11787.932,E2 -11787.932} C_VEL
LIN {X 0,Y 389.68,Z 499.729,A -85,B 0,C 180,E1 -11789.742,E2 -11789.742} C_VEL
LIN {X 0,Y 390.255,Z 493.072,A -85,B 0,C 180,E1 -11791.291,E2 -11791.291} C_VEL
LIN {X 0,Y 390.875,Z 484.837,A -85,B 0,C 180,E1 -11792.835,E2 -11792.835} C_VEL
LIN {X 0,Y 391.545,Z 476.365,A -85,B 0,C 180,E1 -11794.118,E2 -11794.118} C_VEL
LIN {X 0,Y 392.319,Z 465.929,A -85,B 0,C 180,E1 -11795.397,E2 -11795.397} C_VEL
LIN {X 0,Y 393.097,Z 455.578,A -85,B 0,C 180,E1 -11796.416,E2 -11796.416} C_VEL
LIN {X 0,Y 393.837,Z 444.211,A -85,B 0,C 180,E1 -11797.305,E2 -11797.305} C_VEL
LIN {X 0,Y 393.871,Z 442.689,A -85,B 0,C 180,E1 -11797.406,E2 -11797.406} C_VEL
LIN {X 0,Y 393.445,Z 437.326,A -85,B 0,C 180,E1 -11797.768,E2 -11797.768} C_VEL
LIN {X 0,Y 391.024,Z 428.522,A -85,B 0,C 180,E1 -11798.34,E2 -11798.34} C_VEL
LIN {X 0,Y 388.597,Z 419.494,A -85,B 0,C 180,E1 -11798.811,E2 -11798.811} C_VEL
LIN {X 0,Y 388.096,Z 413.791,A -85,B 0,C 180,E1 -11799.012,E2 -11799.012} C_VEL
LIN {X 0,Y 388.866,Z 365.102,A -85,B 0,C 180,E1 -11799.936,E2 -11799.936} C_VEL
LIN {X 0,Y 389.348,Z 327.055,A -85,B 0,C 180,E1 -11800.636,E2 -11800.636} C_VEL
LIN {X 0,Y 386.087,Z 310.469,A -85,B 0,C 180,E1 -11801.103,E2 -11801.103} C_VEL
LIN {X 0,Y 384.519,Z 305.18,A -85,B 0,C 180,E1 -11801.311,E2 -11801.311} C_VEL
LIN {X 0,Y 383.182,Z 297.754,A -85,B 0,C 180,E1 -11803.171,E2 -11803.171} C_VEL
LIN {X 0,Y 383.1,Z 297.763,A -85,B 0,C 180,E1 -11807.07,E2 -11807.07} C_VEL
LIN {X 0,Y 383.035,Z 297.774,A -85,B 0,C 180,E1 -11810.647,E2 -11810.647} C_VEL
LIN {X 0,Y 383.015,Z 297.771,A -85,B 0,C 180,E1 -11813.809,E2 -11813.809} C_VEL
LIN {X 0,Y 382.975,Z 297.779,A -85,B 0,C 180,E1 -11817.309,E2 -11817.309} C_VEL
LIN {X 0,Y 382.986,Z 297.781,A -85,B 0,C 180,E1 -11820.919,E2 -11820.919} C_VEL
LIN {X 0,Y 383.022,Z 297.772,A -85,B 0,C 180,E1 -11824.668,E2 -11824.668} C_VEL
LIN {X 0,Y 382.999,Z 297.773,A -85,B 0,C 180,E1 -11827.903,E2 -11827.903} C_VEL
LIN {X 0,Y 382.965,Z 297.783,A -85,B 0,C 180,E1 -11831.351,E2 -11831.351} C_VEL
LIN {X 0,Y 382.994,Z 297.773,A -85,B 0,C 180,E1 -11834.302,E2 -11834.302} C_VEL
LIN {X 0,Y 383.016,Z 297.776,A -85,B 0,C 180,E1 -11837.24,E2 -11837.24} C_VEL
LIN {X 0,Y 382.99,Z 297.774,A -85,B 0,C 180,E1 -11840.419,E2 -11840.419} C_VEL
LIN {X 0,Y 383.019,Z 297.772,A -85,B 0,C 180,E1 -11844.043,E2 -11844.043} C_VEL
LIN {X 0,Y 382.991,Z 297.781,A -85,B 0,C 180,E1 -11847.578,E2 -11847.578} C_VEL
LIN {X 0,Y 382.985,Z 297.775,A -85,B 0,C 180,E1 -11850.299,E2 -11850.299} C_VEL
LIN {X 0,Y 383.009,Z 297.775,A -85,B 0,C 180,E1 -11854.044,E2 -11854.044} C_VEL
LIN {X 0,Y 382.994,Z 297.775,A -85,B 0,C 180,E1 -11857.334,E2 -11857.334} C_VEL
LIN {X 0,Y 383.063,Z 297.765,A -85,B 0,C 180,E1 -11860.716,E2 -11860.716} C_VEL
LIN {X 0,Y 383.085,Z 297.768,A -85,B 0,C 180,E1 -11864.026,E2 -11864.026} C_VEL
LIN {X 0,Y 383.139,Z 297.756,A -85,B 0,C 180,E1 -11867.284,E2 -11867.284} C_VEL
LIN {X 0,Y 383.141,Z 297.757,A -85,B 0,C 180,E1 -11870.497,E2 -11870.497} C_VEL
LIN {X 0,Y 383.243,Z 297.744,A -85,B 0,C 180,E1 -11873.683,E2 -11873.683} C_VEL
LIN {X 0,Y 383.377,Z 297.729,A -85,B 0,C 180,E1 -11877.899,E2 -11877.899} C_VEL
LIN {X 0,Y 383.376,Z 297.73,A -85,B 0,C 180,E1 -11882.101,E2 -11882.101} C_VEL
LIN {X 0,Y 383.237,Z 297.749,A -85,B 0,C 180,E1 -11886.317,E2 -11886.317} C_VEL
LIN {X 0,Y 383.139,Z 297.755,A -85,B 0,C 180,E1 -11889.502,E2 -11889.502} C_VEL
LIN {X 0,Y 383.13,Z 297.756,A -85,B 0,C 180,E1 -11893.536,E2 -11893.536} C_VEL
LIN {X 0,Y 383.08,Z 297.763,A -85,B 0,C 180,E1 -11897.445,E2 -11897.445} C_VEL
LIN {X 0,Y 383.033,Z 297.775,A -85,B 0,C 180,E1 -11900.646,E2 -11900.646} C_VEL
LIN {X 0,Y 383.013,Z 297.771,A -85,B 0,C 180,E1 -11903.809,E2 -11903.809} C_VEL
LIN {X 0,Y 382.972,Z 297.778,A -85,B 0,C 180,E1 -11907.308,E2 -11907.308} C_VEL
LIN {X 0,Y 382.984,Z 297.781,A -85,B 0,C 180,E1 -11910.918,E2 -11910.918} C_VEL
LIN {X 0,Y 383.014,Z 297.774,A -85,B 0,C 180,E1 -11914.668,E2 -11914.668} C_VEL
LIN {X 0,Y 382.997,Z 297.773,A -85,B 0,C 180,E1 -11917.902,E2 -11917.902} C_VEL
LIN {X 0,Y 382.963,Z 297.783,A -85,B 0,C 180,E1 -11921.35,E2 -11921.35} C_VEL
LIN {X 0,Y 382.992,Z 297.774,A -85,B 0,C 180,E1 -11924.302,E2 -11924.302} C_VEL
LIN {X 0,Y 383.013,Z 297.777,A -85,B 0,C 180,E1 -11927.24,E2 -11927.24} C_VEL
LIN {X 0,Y 382.987,Z 297.774,A -85,B 0,C 180,E1 -11930.419,E2 -11930.419} C_VEL
LIN {X 0,Y 383.016,Z 297.772,A -85,B 0,C 180,E1 -11934.043,E2 -11934.043} C_VEL
LIN {X 0,Y 382.988,Z 297.781,A -85,B 0,C 180,E1 -11937.578,E2 -11937.578} C_VEL
LIN {X 0,Y 383.068,Z 297.793,A -85,B 0,C 180,E1 -11941.134,E2 -11941.134} C_VEL
LIN {X 0,Y 385.947,Z 312.325,A -85,B 0,C 180,E1 -11944.374,E2 -11944.374} C_VEL
LIN {X 0,Y 386.173,Z 316.497,A -85,B 0,C 180,E1 -11945.254,E2 -11945.254} C_VEL
LIN {X 0,Y 384.786,Z 335.656,A -85,B 0,C 180,E1 -11949.135,E2 -11949.135} C_VEL
LIN {X 0,Y 384.603,Z 338.922,A -85,B 0,C 180,E1 -11949.745,E2 -11949.745} C_VEL
LIN {X 0,Y 388.975,Z 371.072,A -85,B 0,C 180,E1 -11950.553,E2 -11950.553} C_VEL
LIN {X 0,Y 387.965,Z 448.031,A -85,B 0,C 180,E1 -11951.995,E2 -11951.995} C_VEL
LIN {X 0,Y 387.297,Z 461.893,A -85,B 0,C 180,E1 -11952.475,E2 -11952.475} C_VEL
LIN {X 0,Y 386.558,Z 474.845,A -85,B 0,C 180,E1 -11953.156,E2 -11953.156} C_VEL
LIN {X 0,Y 385.734,Z 486.658,A -85,B 0,C 180,E1 -11954.003,E2 -11954.003} C_VEL
LIN {X 0,Y 384.863,Z 498.053,A -85,B 0,C 180,E1 -11955.052,E2 -11955.052} C_VEL
LIN {X 0,Y 384.173,Z 508.323,A -85,B 0,C 180,E1 -11956.241,E2 -11956.241} C_VEL
LIN {X 0,Y 383.389,Z 517.545,A -85,B 0,C 180,E1 -11957.561,E2 -11957.561} C_VEL
LIN {X 0,Y 382.624,Z 526.526,A -85,B 0,C 180,E1 -11959.147,E2 -11959.147} C_VEL
LIN {X 0,Y 382.153,Z 533.744,A -85,B 0,C 180,E1 -11960.739,E2 -11960.739} C_VEL
LIN {X 0,Y 381.849,Z 540.308,A -85,B 0,C 180,E1 -11962.597,E2 -11962.597} C_VEL
LIN {X 0,Y 381.704,Z 543.855,A -85,B 0,C 180,E1 -11963.858,E2 -11963.858} C_VEL
LIN {X 0,Y 381.638,Z 547.882,A -85,B 0,C 180,E1 -11965.775,E2 -11965.775} C_VEL
LIN {X 0,Y 381.688,Z 550.696,A -85,B 0,C 180,E1 -11967.889,E2 -11967.889} C_VEL
LIN {X 0,Y 381.692,Z 551.448,A -85,B 0,C 180,E1 -11968.944,E2 -11968.944} C_VEL
LIN {X 0,Y 381.691,Z 551.767,A -85,B 0,C 180,E1 -11971.054,E2 -11971.054} C_VEL
LIN {X 0,Y 381.653,Z 551.343,A -85,B 0,C 180,E1 -11972.11,E2 -11972.11} C_VEL
LIN {X 0,Y 381.579,Z 550.486,A -85,B 0,C 180,E1 -11973.167,E2 -11973.167} C_VEL
LIN {X 0,Y 381.63,Z 549.224,A -85,B 0,C 180,E1 -11974.224,E2 -11974.224} C_VEL
LIN {X 0,Y 381.677,Z 545.961,A -85,B 0,C 180,E1 -11976.105,E2 -11976.105} C_VEL
LIN {X 0,Y 381.939,Z 541.443,A -85,B 0,C 180,E1 -11977.932,E2 -11977.932} C_VEL
LIN {X 0,Y 382.401,Z 535.271,A -85,B 0,C 180,E1 -11979.787,E2 -11979.787} C_VEL
LIN {X 0,Y 383.018,Z 528.565,A -85,B 0,C 180,E1 -11981.376,E2 -11981.376} C_VEL
LIN {X 0,Y 383.994,Z 520.273,A -85,B 0,C 180,E1 -11982.955,E2 -11982.955} C_VEL
LIN {X 0,Y 384.952,Z 510.454,A -85,B 0,C 180,E1 -11984.453,E2 -11984.453} C_VEL
LIN {X 0,Y 386.031,Z 500.16,A -85,B 0,C 180,E1 -11985.712,E2 -11985.712} C_VEL
LIN {X 0,Y 387.112,Z 489.591,A -85,B 0,C 180,E1 -11986.75,E2 -11986.75} C_VEL
LIN {X 0,Y 388.232,Z 477.833,A -85,B 0,C 180,E1 -11987.65,E2 -11987.65} C_VEL
LIN {X 0,Y 389.065,Z 466.936,A -85,B 0,C 180,E1 -11988.291,E2 -11988.291} C_VEL
LIN {X 0,Y 389.934,Z 453.223,A -85,B 0,C 180,E1 -11988.862,E2 -11988.862} C_VEL
LIN {X 0,Y 390.375,Z 440.259,A -85,B 0,C 180,E1 -11989.191,E2 -11989.191} C_VEL
LIN {X 0,Y 391.294,Z 370.651,A -85,B 0,C 180,E1 -11990.495,E2 -11990.495} C_VEL
LIN {X 0,Y 387.927,Z 349.877,A -85,B 0,C 180,E1 -11991.118,E2 -11991.118} C_VEL
LIN {X 0,Y 385.688,Z 338.089,A -85,B 0,C 180,E1 -11991.516,E2 -11991.516} C_VEL
LIN {X 0,Y 387.202,Z 321.573,A -85,B 0,C 180,E1 -11994.932,E2 -11994.932} C_VEL
LIN {X 0,Y 387.28,Z 317.438,A -85,B 0,C 180,E1 -11995.818,E2 -11995.818} C_VEL
LIN {X 0,Y 385.138,Z 306.749,A -85,B 0,C 180,E1 -11998.323,E2 -11998.323} C_VEL
LIN {X 0,Y 382.977,Z 297.791,A -85,B 0,C 180,E1 -12000.566,E2 -12000.566} C_VEL
LIN {X 0,Y 383.001,Z 297.784,A -85,B 0,C 180,E1 -12003.4,E2 -12003.4} C_VEL
LIN {X 0,Y 383.029,Z 297.777,A -85,B 0,C 180,E1 -12006.164,E2 -12006.164} C_VEL
LIN {X 0,Y 383.005,Z 297.775,A -85,B 0,C 180,E1 -12009.958,E2 -12009.958} C_VEL
LIN {X 0,Y 383.002,Z 297.777,A -85,B 0,C 180,E1 -12012.778,E2 -12012.778} C_VEL
LIN {X 0,Y 382.994,Z 297.776,A -85,B 0,C 180,E1 -12015.789,E2 -12015.789} C_VEL
LIN {X 0,Y 382.985,Z 297.776,A -85,B 0,C 180,E1 -12018.795,E2 -12018.795} C_VEL
LIN {X 0,Y 382.997,Z 297.773,A -85,B 0,C 180,E1 -12022.096,E2 -12022.096} C_VEL
LIN {X 0,Y 383.014,Z 297.768,A -85,B 0,C 180,E1 -12025.332,E2 -12025.332} C_VEL
LIN {X 0,Y 382.979,Z 297.776,A -85,B 0,C 180,E1 -12029.081,E2 -12029.081} C_VEL
LIN {X 0,Y 383.053,Z 297.767,A -85,B 0,C 180,E1 -12032.698,E2 -12032.698} C_VEL
LIN {X 0,Y 383.048,Z 297.765,A -85,B 0,C 180,E1 -12035.04,E2 -12035.04} C_VEL
LIN {X 0,Y 382.995,Z 297.778,A -85,B 0,C 180,E1 -12038.469,E2 -12038.469} C_VEL
LIN {X 0,Y 383.059,Z 297.766,A -85,B 0,C 180,E1 -12041.826,E2 -12041.826} C_VEL
LIN {X 0,Y 383.107,Z 297.764,A -85,B 0,C 180,E1 -12045.118,E2 -12045.118} C_VEL
LIN {X 0,Y 383.094,Z 297.758,A -85,B 0,C 180,E1 -12048.358,E2 -12048.358} C_VEL
LIN {X 0,Y 383.3,Z 297.731,A -85,B 0,C 180,E1 -12051.933,E2 -12051.933} C_VEL
LIN {X 0,Y 383.196,Z 297.755,A -85,B 0,C 180,E1 -12054.739,E2 -12054.739} C_VEL
LIN {X 0,Y 383.385,Z 297.725,A -85,B 0,C 180,E1 -12057.899,E2 -12057.899} C_VEL
LIN {X 0,Y 383.516,Z 297.706,A -85,B 0,C 180,E1 -12060,E2 -12060} C_VEL
LIN {X 0,Y 383.247,Z 297.745,A -85,B 0,C 180,E1 -12063.154,E2 -12063.154} C_VEL
LIN {X 0,Y 383.266,Z 297.738,A -85,B 0,C 180,E1 -12066.637,E2 -12066.637} C_VEL
LIN {X 0,Y 383.257,Z 297.741,A -85,B 0,C 180,E1 -12068.436,E2 -12068.436} C_VEL
LIN {X 0,Y 383.095,Z 297.762,A -85,B 0,C 180,E1 -12071.643,E2 -12071.643} C_VEL
LIN {X 0,Y 383.107,Z 297.762,A -85,B 0,C 180,E1 -12074.882,E2 -12074.882} C_VEL
LIN {X 0,Y 383.059,Z 297.763,A -85,B 0,C 180,E1 -12078.174,E2 -12078.174} C_VEL
LIN {X 0,Y 382.99,Z 297.774,A -85,B 0,C 180,E1 -12081.532,E2 -12081.532} C_VEL
LIN {X 0,Y 383.049,Z 297.769,A -85,B 0,C 180,E1 -12084.961,E2 -12084.961} C_VEL
LIN {X 0,Y 383.027,Z 297.769,A -85,B 0,C 180,E1 -12088.271,E2 -12088.271} C_VEL
LIN {X 0,Y 383.007,Z 297.768,A -85,B 0,C 180,E1 -12092.15,E2 -12092.15} C_VEL
LIN {X 0,Y 383.016,Z 297.772,A -85,B 0,C 180,E1 -12094.669,E2 -12094.669} C_VEL
LIN {X 0,Y 382.993,Z 297.771,A -85,B 0,C 180,E1 -12097.904,E2 -12097.904} C_VEL
LIN {X 0,Y 382.965,Z 297.78,A -85,B 0,C 180,E1 -12101.351,E2 -12101.351} C_VEL
LIN {X 0,Y 382.993,Z 297.776,A -85,B 0,C 180,E1 -12104.304,E2 -12104.304} C_VEL
LIN {X 0,Y 383.01,Z 297.777,A -85,B 0,C 180,E1 -12107.241,E2 -12107.241} C_VEL
LIN {X 0,Y 382.985,Z 297.778,A -85,B 0,C 180,E1 -12110.42,E2 -12110.42} C_VEL
LIN {X 0,Y 383.023,Z 297.771,A -85,B 0,C 180,E1 -12114.045,E2 -12114.045} C_VEL
LIN {X 0,Y 383.031,Z 297.847,A -85,B 0,C 180,E1 -12117.439,E2 -12117.439} C_VEL
LIN {X 0,Y 384.898,Z 305.918,A -85,B 0,C 180,E1 -12119.486,E2 -12119.486} C_VEL
LIN {X 0,Y 389.599,Z 317.828,A -85,B 0,C 180,E1 -12120.041,E2 -12120.041} C_VEL
LIN {X 0,Y 392.011,Z 328.253,A -85,B 0,C 180,E1 -12120.404,E2 -12120.404} C_VEL
LIN {X 0,Y 390.527,Z 413.543,A -85,B 0,C 180,E1 -12122.014,E2 -12122.014} C_VEL
LIN {X 0,Y 390.111,Z 426.511,A -85,B 0,C 180,E1 -12122.471,E2 -12122.471} C_VEL
LIN {X 0,Y 389.363,Z 438.87,A -85,B 0,C 180,E1 -12123.104,E2 -12123.104} C_VEL
LIN {X 0,Y 388.598,Z 449.585,A -85,B 0,C 180,E1 -12123.844,E2 -12123.844} C_VEL
LIN {X 0,Y 387.783,Z 459.936,A -85,B 0,C 180,E1 -12124.753,E2 -12124.753} C_VEL
LIN {X 0,Y 386.643,Z 471.231,A -85,B 0,C 180,E1 -12126.002,E2 -12126.002} C_VEL
LIN {X 0,Y 385.699,Z 480.111,A -85,B 0,C 180,E1 -12127.22,E2 -12127.22} C_VEL
LIN {X 0,Y 384.732,Z 488.869,A -85,B 0,C 180,E1 -12128.692,E2 -12128.692} C_VEL
LIN {X 0,Y 383.874,Z 496.108,A -85,B 0,C 180,E1 -12130.203,E2 -12130.203} C_VEL
LIN {X 0,Y 383.125,Z 502.36,A -85,B 0,C 180,E1 -12131.83,E2 -12131.83} C_VEL
LIN {X 0,Y 382.603,Z 507.287,A -85,B 0,C 180,E1 -12133.459,E2 -12133.459} C_VEL
LIN {X 0,Y 382.194,Z 511.046,A -85,B 0,C 180,E1 -12135.082,E2 -12135.082} C_VEL
LIN {X 0,Y 381.962,Z 512.973,A -85,B 0,C 180,E1 -12136.162,E2 -12136.162} C_VEL
LIN {X 0,Y 381.88,Z 514.477,A -85,B 0,C 180,E1 -12137.267,E2 -12137.267} C_VEL
LIN {X 0,Y 381.628,Z 516.113,A -85,B 0,C 180,E1 -12139.389,E2 -12139.389} C_VEL
LIN {X 0,Y 381.589,Z 516.358,A -85,B 0,C 180,E1 -12140.459,E2 -12140.459} C_VEL
LIN {X 0,Y 381.6,Z 516.185,A -85,B 0,C 180,E1 -12141.528,E2 -12141.528} C_VEL
LIN {X 0,Y 381.661,Z 515.593,A -85,B 0,C 180,E1 -12142.595,E2 -12142.595} C_VEL
LIN {X 0,Y 381.755,Z 514.475,A -85,B 0,C 180,E1 -12143.792,E2 -12143.792} C_VEL
LIN {X 0,Y 381.822,Z 511.444,A -85,B 0,C 180,E1 -12145.778,E2 -12145.778} C_VEL
LIN {X 0,Y 382.126,Z 507.898,A -85,B 0,C 180,E1 -12147.365,E2 -12147.365} C_VEL
LIN {X 0,Y 382.326,Z 503.277,A -85,B 0,C 180,E1 -12148.947,E2 -12148.947} C_VEL
LIN {X 0,Y 383.017,Z 496.289,A -85,B 0,C 180,E1 -12150.789,E2 -12150.789} C_VEL
LIN {X 0,Y 383.592,Z 488.753,A -85,B 0,C 180,E1 -12152.363,E2 -12152.363} C_VEL
LIN {X 0,Y 384.387,Z 479.277,A -85,B 0,C 180,E1 -12153.932,E2 -12153.932} C_VEL
LIN {X 0,Y 385.136,Z 469.518,A -85,B 0,C 180,E1 -12155.236,E2 -12155.236} C_VEL
LIN {X 0,Y 385.977,Z 458.569,A -85,B 0,C 180,E1 -12156.404,E2 -12156.404} C_VEL
LIN {X 0,Y 386.854,Z 446.094,A -85,B 0,C 180,E1 -12157.438,E2 -12157.438} C_VEL
LIN {X 0,Y 387.367,Z 433.83,A -85,B 0,C 180,E1 -12158.215,E2 -12158.215} C_VEL
LIN {X 0,Y 387.898,Z 420.705,A -85,B 0,C 180,E1 -12158.794,E2 -12158.794} C_VEL
LIN {X 0,Y 388.096,Z 413.791,A -85,B 0,C 180,E1 -12159.012,E2 -12159.012} C_VEL
LIN {X 0,Y 387.608,Z 408.021,A -85,B 0,C 180,E1 -12159.185,E2 -12159.185} C_VEL
LIN {X 0,Y 382.328,Z 389.293,A -85,B 0,C 180,E1 -12159.766,E2 -12159.766} C_VEL
LIN {X 0,Y 381.773,Z 383.473,A -85,B 0,C 180,E1 -12159.896,E2 -12159.896} C_VEL
LIN {X 0,Y 382.515,Z 327.586,A -85,B 0,C 180,E1 -12160.942,E2 -12160.942} C_VEL
LIN {X 0,Y 379.562,Z 312.584,A -85,B 0,C 180,E1 -12161.374,E2 -12161.374} C_VEL
LIN {X 0,Y 377.401,Z 305.569,A -85,B 0,C 180,E1 -12161.636,E2 -12161.636} C_VEL
LIN {X 0,Y 376.125,Z 298.632,A -85,B 0,C 180,E1 -12163.407,E2 -12163.407} C_VEL
LIN {X 0,Y 376.031,Z 298.643,A -85,B 0,C 180,E1 -12166.282,E2 -12166.282} C_VEL
LIN {X 0,Y 376.002,Z 298.644,A -85,B 0,C 180,E1 -12169.661,E2 -12169.661} C_VEL
LIN {X 0,Y 375.979,Z 298.647,A -85,B 0,C 180,E1 -12173.66,E2 -12173.66} C_VEL
LIN {X 0,Y 375.918,Z 298.659,A -85,B 0,C 180,E1 -12176.661,E2 -12176.661} C_VEL
LIN {X 0,Y 375.918,Z 298.66,A -85,B 0,C 180,E1 -12179.084,E2 -12179.084} C_VEL
LIN {X 0,Y 375.961,Z 298.651,A -85,B 0,C 180,E1 -12181.562,E2 -12181.562} C_VEL
LIN {X 0,Y 375.961,Z 298.653,A -85,B 0,C 180,E1 -12185.416,E2 -12185.416} C_VEL
LIN {X 0,Y 375.941,Z 298.652,A -85,B 0,C 180,E1 -12188.263,E2 -12188.263} C_VEL
LIN {X 0,Y 375.92,Z 298.658,A -85,B 0,C 180,E1 -12191.597,E2 -12191.597} C_VEL
LIN {X 0,Y 375.926,Z 298.655,A -85,B 0,C 180,E1 -12194.73,E2 -12194.73} C_VEL
LIN {X 0,Y 375.93,Z 298.657,A -85,B 0,C 180,E1 -12197.699,E2 -12197.699} C_VEL
LIN {X 0,Y 375.939,Z 298.652,A -85,B 0,C 180,E1 -12200.534,E2 -12200.534} C_VEL
LIN {X 0,Y 375.963,Z 298.657,A -85,B 0,C 180,E1 -12203.497,E2 -12203.497} C_VEL
LIN {X 0,Y 375.962,Z 298.652,A -85,B 0,C 180,E1 -12205.888,E2 -12205.888} C_VEL
LIN {X 0,Y 375.967,Z 298.655,A -85,B 0,C 180,E1 -12209.687,E2 -12209.687} C_VEL
LIN {X 0,Y 375.938,Z 298.654,A -85,B 0,C 180,E1 -12212.136,E2 -12212.136} C_VEL
LIN {X 0,Y 375.964,Z 298.656,A -85,B 0,C 180,E1 -12215.716,E2 -12215.716} C_VEL
LIN {X 0,Y 376.003,Z 298.645,A -85,B 0,C 180,E1 -12219.198,E2 -12219.198} C_VEL
LIN {X 0,Y 376.037,Z 298.641,A -85,B 0,C 180,E1 -12222.6,E2 -12222.6} C_VEL
LIN {X 0,Y 376.094,Z 298.636,A -85,B 0,C 180,E1 -12226.342,E2 -12226.342} C_VEL
LIN {X 0,Y 376.112,Z 298.635,A -85,B 0,C 180,E1 -12230.318,E2 -12230.318} C_VEL
LIN {X 0,Y 376.202,Z 298.621,A -85,B 0,C 180,E1 -12233.564,E2 -12233.564} C_VEL
LIN {X 0,Y 376.342,Z 298.605,A -85,B 0,C 180,E1 -12237.859,E2 -12237.859} C_VEL
LIN {X 0,Y 376.341,Z 298.607,A -85,B 0,C 180,E1 -12242.14,E2 -12242.14} C_VEL
LIN {X 0,Y 376.197,Z 298.627,A -85,B 0,C 180,E1 -12246.436,E2 -12246.436} C_VEL
LIN {X 0,Y 376.11,Z 298.631,A -85,B 0,C 180,E1 -12249.681,E2 -12249.681} C_VEL
LIN {X 0,Y 376.094,Z 298.633,A -85,B 0,C 180,E1 -12253.657,E2 -12253.657} C_VEL
LIN {X 0,Y 376.031,Z 298.641,A -85,B 0,C 180,E1 -12257.599,E2 -12257.599} C_VEL
LIN {X 0,Y 375.982,Z 298.653,A -85,B 0,C 180,E1 -12260.832,E2 -12260.832} C_VEL
LIN {X 0,Y 375.972,Z 298.65,A -85,B 0,C 180,E1 -12264.283,E2 -12264.283} C_VEL
LIN {X 0,Y 375.92,Z 298.654,A -85,B 0,C 180,E1 -12267.865,E2 -12267.865} C_VEL
LIN {X 0,Y 375.957,Z 298.654,A -85,B 0,C 180,E1 -12270.693,E2 -12270.693} C_VEL
LIN {X 0,Y 375.96,Z 298.65,A -85,B 0,C 180,E1 -12274.111,E2 -12274.111} C_VEL
LIN {X 0,Y 375.952,Z 298.654,A -85,B 0,C 180,E1 -12276.741,E2 -12276.741} C_VEL
LIN {X 0,Y 375.941,Z 298.652,A -85,B 0,C 180,E1 -12279.961,E2 -12279.961} C_VEL
LIN {X 0,Y 375.928,Z 298.655,A -85,B 0,C 180,E1 -12283.766,E2 -12283.766} C_VEL
LIN {X 0,Y 375.934,Z 298.655,A -85,B 0,C 180,E1 -12286.811,E2 -12286.811} C_VEL
LIN {X 0,Y 375.936,Z 298.653,A -85,B 0,C 180,E1 -12290.533,E2 -12290.533} C_VEL
LIN {X 0,Y 375.96,Z 298.656,A -85,B 0,C 180,E1 -12293.496,E2 -12293.496} C_VEL
LIN {X 0,Y 375.96,Z 298.652,A -85,B 0,C 180,E1 -12295.888,E2 -12295.888} C_VEL
LIN {X 0,Y 375.966,Z 298.656,A -85,B 0,C 180,E1 -12299.687,E2 -12299.687} C_VEL
LIN {X 0,Y 375.995,Z 298.695,A -85,B 0,C 180,E1 -12300.884,E2 -12300.884} C_VEL
LIN {X 0,Y 378.862,Z 313.061,A -85,B 0,C 180,E1 -12304.155,E2 -12304.155} C_VEL
LIN {X 0,Y 379.233,Z 317.418,A -85,B 0,C 180,E1 -12305.098,E2 -12305.098} C_VEL
LIN {X 0,Y 377.78,Z 336.62,A -85,B 0,C 180,E1 -12309.059,E2 -12309.059} C_VEL
LIN {X 0,Y 377.643,Z 338.331,A -85,B 0,C 180,E1 -12309.408,E2 -12309.408} C_VEL
LIN {X 0,Y 382.153,Z 372.79,A -85,B 0,C 180,E1 -12310.286,E2 -12310.286} C_VEL
LIN {X 0,Y 381.102,Z 447.07,A -85,B 0,C 180,E1 -12311.694,E2 -12311.694} C_VEL
LIN {X 0,Y 380.516,Z 460.386,A -85,B 0,C 180,E1 -12312.152,E2 -12312.152} C_VEL
LIN {X 0,Y 379.837,Z 472.606,A -85,B 0,C 180,E1 -12312.779,E2 -12312.779} C_VEL
LIN {X 0,Y 378.998,Z 484.106,A -85,B 0,C 180,E1 -12313.573,E2 -12313.573} C_VEL
LIN {X 0,Y 378.036,Z 495.913,A -85,B 0,C 180,E1 -12314.637,E2 -12314.637} C_VEL
LIN {X 0,Y 377.256,Z 505.995,A -85,B 0,C 180,E1 -12315.779,E2 -12315.779} C_VEL
LIN {X 0,Y 376.489,Z 515.185,A -85,B 0,C 180,E1 -12317.055,E2 -12317.055} C_VEL
LIN {X 0,Y 375.862,Z 523.169,A -85,B 0,C 180,E1 -12318.403,E2 -12318.403} C_VEL
LIN {X 0,Y 375.255,Z 530.952,A -85,B 0,C 180,E1 -12320.023,E2 -12320.023} C_VEL
LIN {X 0,Y 374.842,Z 538.115,A -85,B 0,C 180,E1 -12321.916,E2 -12321.916} C_VEL
LIN {X 0,Y 374.632,Z 542.871,A -85,B 0,C 180,E1 -12323.536,E2 -12323.536} C_VEL
LIN {X 0,Y 374.57,Z 546.498,A -85,B 0,C 180,E1 -12325.156,E2 -12325.156} C_VEL
LIN {X 0,Y 374.509,Z 549.093,A -85,B 0,C 180,E1 -12326.772,E2 -12326.772} C_VEL
LIN {X 0,Y 374.588,Z 550.317,A -85,B 0,C 180,E1 -12327.849,E2 -12327.849} C_VEL
LIN {X 0,Y 374.625,Z 551.096,A -85,B 0,C 180,E1 -12328.924,E2 -12328.924} C_VEL
LIN {X 0,Y 374.622,Z 551.444,A -85,B 0,C 180,E1 -12331.074,E2 -12331.074} C_VEL
LIN {X 0,Y 374.552,Z 551.035,A -85,B 0,C 180,E1 -12332.15,E2 -12332.15} C_VEL
LIN {X 0,Y 374.491,Z 550.207,A -85,B 0,C 180,E1 -12333.227,E2 -12333.227} C_VEL
LIN {X 0,Y 374.555,Z 548.96,A -85,B 0,C 180,E1 -12334.304,E2 -12334.304} C_VEL
LIN {X 0,Y 374.573,Z 546.063,A -85,B 0,C 180,E1 -12336.053,E2 -12336.053} C_VEL
LIN {X 0,Y 374.876,Z 541.247,A -85,B 0,C 180,E1 -12338.082,E2 -12338.082} C_VEL
LIN {X 0,Y 375.376,Z 535.13,A -85,B 0,C 180,E1 -12339.972,E2 -12339.972} C_VEL
LIN {X 0,Y 376.016,Z 528.467,A -85,B 0,C 180,E1 -12341.59,E2 -12341.59} C_VEL
LIN {X 0,Y 377.062,Z 520.224,A -85,B 0,C 180,E1 -12343.198,E2 -12343.198} C_VEL
LIN {X 0,Y 377.994,Z 511.184,A -85,B 0,C 180,E1 -12344.628,E2 -12344.628} C_VEL
LIN {X 0,Y 379.2,Z 500.284,A -85,B 0,C 180,E1 -12346.002,E2 -12346.002} C_VEL
LIN {X 0,Y 380.315,Z 489.815,A -85,B 0,C 180,E1 -12347.059,E2 -12347.059} C_VEL
LIN {X 0,Y 381.508,Z 478.278,A -85,B 0,C 180,E1 -12347.972,E2 -12347.972} C_VEL
LIN {X 0,Y 382.374,Z 467.624,A -85,B 0,C 180,E1 -12348.623,E2 -12348.623} C_VEL
LIN {X 0,Y 383.263,Z 454.329,A -85,B 0,C 180,E1 -12349.203,E2 -12349.203} C_VEL
LIN {X 0,Y 383.793,Z 440.697,A -85,B 0,C 180,E1 -12349.573,E2 -12349.573} C_VEL
LIN {X 0,Y 384.784,Z 371.632,A -85,B 0,C 180,E1 -12350.887,E2 -12350.887} C_VEL
LIN {X 0,Y 381.652,Z 352.154,A -85,B 0,C 180,E1 -12351.485,E2 -12351.485} C_VEL
LIN {X 0,Y 378.889,Z 337.747,A -85,B 0,C 180,E1 -12351.981,E2 -12351.981} C_VEL
LIN {X 0,Y 380.352,Z 322.715,A -85,B 0,C 180,E1 -12355.149,E2 -12355.149} C_VEL
LIN {X 0,Y 380.35,Z 318.713,A -85,B 0,C 180,E1 -12356.03,E2 -12356.03} C_VEL
LIN {X 0,Y 378.213,Z 308.033,A -85,B 0,C 180,E1 -12358.586,E2 -12358.586} C_VEL
LIN {X 0,Y 375.942,Z 298.664,A -85,B 0,C 180,E1 -12360.951,E2 -12360.951} C_VEL
LIN {X 0,Y 375.977,Z 298.658,A -85,B 0,C 180,E1 -12364.667,E2 -12364.667} C_VEL
LIN {X 0,Y 375.969,Z 298.656,A -85,B 0,C 180,E1 -12368.269,E2 -12368.269} C_VEL
LIN {X 0,Y 375.931,Z 298.653,A -85,B 0,C 180,E1 -12371.6,E2 -12371.6} C_VEL
LIN {X 0,Y 375.924,Z 298.657,A -85,B 0,C 180,E1 -12375.268,E2 -12375.268} C_VEL
LIN {X 0,Y 375.931,Z 298.657,A -85,B 0,C 180,E1 -12378.399,E2 -12378.399} C_VEL
LIN {X 0,Y 375.971,Z 298.648,A -85,B 0,C 180,E1 -12381.729,E2 -12381.729} C_VEL
LIN {X 0,Y 375.976,Z 298.645,A -85,B 0,C 180,E1 -12385.332,E2 -12385.332} C_VEL
LIN {X 0,Y 375.954,Z 298.65,A -85,B 0,C 180,E1 -12388.438,E2 -12388.438} C_VEL
LIN {X 0,Y 375.979,Z 298.645,A -85,B 0,C 180,E1 -12392.14,E2 -12392.14} C_VEL
LIN {X 0,Y 376.003,Z 298.648,A -85,B 0,C 180,E1 -12394.539,E2 -12394.539} C_VEL
LIN {X 0,Y 375.964,Z 298.65,A -85,B 0,C 180,E1 -12398.046,E2 -12398.046} C_VEL
LIN {X 0,Y 376.005,Z 298.646,A -85,B 0,C 180,E1 -12401.473,E2 -12401.473} C_VEL
LIN {X 0,Y 376.055,Z 298.642,A -85,B 0,C 180,E1 -12404.833,E2 -12404.833} C_VEL
LIN {X 0,Y 376.046,Z 298.635,A -85,B 0,C 180,E1 -12408.137,E2 -12408.137} C_VEL
LIN {X 0,Y 376.254,Z 298.609,A -85,B 0,C 180,E1 -12411.877,E2 -12411.877} C_VEL
LIN {X 0,Y 376.168,Z 298.629,A -85,B 0,C 180,E1 -12414.64,E2 -12414.64} C_VEL
LIN {X 0,Y 376.351,Z 298.601,A -85,B 0,C 180,E1 -12417.86,E2 -12417.86} C_VEL
LIN {X 0,Y 376.486,Z 298.582,A -85,B 0,C 180,E1 -12420,E2 -12420} C_VEL
LIN {X 0,Y 376.185,Z 298.624,A -85,B 0,C 180,E1 -12423.213,E2 -12423.213} C_VEL
LIN {X 0,Y 376.231,Z 298.615,A -85,B 0,C 180,E1 -12426.628,E2 -12426.628} C_VEL
LIN {X 0,Y 376.202,Z 298.621,A -85,B 0,C 180,E1 -12428.595,E2 -12428.595} C_VEL
LIN {X 0,Y 376.047,Z 298.639,A -85,B 0,C 180,E1 -12431.864,E2 -12431.864} C_VEL
LIN {X 0,Y 376.055,Z 298.644,A -85,B 0,C 180,E1 -12435.168,E2 -12435.168} C_VEL
LIN {X 0,Y 376.006,Z 298.643,A -85,B 0,C 180,E1 -12438.527,E2 -12438.527} C_VEL
LIN {X 0,Y 375.96,Z 298.649,A -85,B 0,C 180,E1 -12441.955,E2 -12441.955} C_VEL
LIN {X 0,Y 376.004,Z 298.645,A -85,B 0,C 180,E1 -12445.462,E2 -12445.462} C_VEL
LIN {X 0,Y 375.959,Z 298.651,A -85,B 0,C 180,E1 -12449.081,E2 -12449.081} C_VEL
LIN {X 0,Y 375.947,Z 298.649,A -85,B 0,C 180,E1 -12452.829,E2 -12452.829} C_VEL
LIN {X 0,Y 375.955,Z 298.651,A -85,B 0,C 180,E1 -12455.416,E2 -12455.416} C_VEL
LIN {X 0,Y 375.936,Z 298.649,A -85,B 0,C 180,E1 -12458.264,E2 -12458.264} C_VEL
LIN {X 0,Y 375.92,Z 298.659,A -85,B 0,C 180,E1 -12461.599,E2 -12461.599} C_VEL
LIN {X 0,Y 375.924,Z 298.658,A -85,B 0,C 180,E1 -12464.732,E2 -12464.732} C_VEL
LIN {X 0,Y 375.925,Z 298.658,A -85,B 0,C 180,E1 -12467.7,E2 -12467.7} C_VEL
LIN {X 0,Y 375.934,Z 298.657,A -85,B 0,C 180,E1 -12470.535,E2 -12470.535} C_VEL
LIN {X 0,Y 375.962,Z 298.656,A -85,B 0,C 180,E1 -12473.497,E2 -12473.497} C_VEL
LIN {X 0,Y 376.001,Z 298.802,A -85,B 0,C 180,E1 -12477.058,E2 -12477.058} C_VEL
LIN {X 0,Y 377.732,Z 306.3,A -85,B 0,C 180,E1 -12478.99,E2 -12478.99} C_VEL
LIN {X 0,Y 383.337,Z 320.019,A -85,B 0,C 180,E1 -12479.664,E2 -12479.664} C_VEL
LIN {X 0,Y 385.586,Z 330.257,A -85,B 0,C 180,E1 -12480.022,E2 -12480.022} C_VEL
LIN {X 0,Y 383.955,Z 413.843,A -85,B 0,C 180,E1 -12481.619,E2 -12481.619} C_VEL
LIN {X 0,Y 383.503,Z 427.27,A -85,B 0,C 180,E1 -12482.104,E2 -12482.104} C_VEL
LIN {X 0,Y 382.719,Z 439.513,A -85,B 0,C 180,E1 -12482.747,E2 -12482.747} C_VEL
LIN {X 0,Y 381.79,Z 451.792,A -85,B 0,C 180,E1 -12483.635,E2 -12483.635} C_VEL
LIN {X 0,Y 380.767,Z 463.558,A -85,B 0,C 180,E1 -12484.746,E2 -12484.746} C_VEL
LIN {X 0,Y 379.62,Z 473.86,A -85,B 0,C 180,E1 -12485.966,E2 -12485.966} C_VEL
LIN {X 0,Y 378.596,Z 483.154,A -85,B 0,C 180,E1 -12487.345,E2 -12487.345} C_VEL
LIN {X 0,Y 377.572,Z 491.437,A -85,B 0,C 180,E1 -12488.856,E2 -12488.856} C_VEL
LIN {X 0,Y 376.744,Z 498.209,A -85,B 0,C 180,E1 -12490.381,E2 -12490.381} C_VEL
LIN {X 0,Y 375.988,Z 504.295,A -85,B 0,C 180,E1 -12492.093,E2 -12492.093} C_VEL
LIN {X 0,Y 375.463,Z 508.731,A -85,B 0,C 180,E1 -12493.694,E2 -12493.694} C_VEL
LIN {X 0,Y 375.187,Z 511.144,A -85,B 0,C 180,E1 -12494.797,E2 -12494.797} C_VEL
LIN {X 0,Y 374.933,Z 513.108,A -85,B 0,C 180,E1 -12495.897,E2 -12495.897} C_VEL
LIN {X 0,Y 374.795,Z 514.853,A -85,B 0,C 180,E1 -12497.185,E2 -12497.185} C_VEL
LIN {X 0,Y 374.545,Z 516.393,A -85,B 0,C 180,E1 -12499.186,E2 -12499.186} C_VEL
LIN {X 0,Y 374.5,Z 516.563,A -85,B 0,C 180,E1 -12501.366,E2 -12501.366} C_VEL
LIN {X 0,Y 374.573,Z 516.013,A -85,B 0,C 180,E1 -12502.454,E2 -12502.454} C_VEL
LIN {X 0,Y 374.685,Z 514.804,A -85,B 0,C 180,E1 -12503.793,E2 -12503.793} C_VEL
LIN {X 0,Y 374.736,Z 512.006,A -85,B 0,C 180,E1 -12505.698,E2 -12505.698} C_VEL
LIN {X 0,Y 375.038,Z 508.535,A -85,B 0,C 180,E1 -12507.315,E2 -12507.315} C_VEL
LIN {X 0,Y 375.252,Z 503.997,A -85,B 0,C 180,E1 -12508.928,E2 -12508.928} C_VEL
LIN {X 0,Y 375.922,Z 497.105,A -85,B 0,C 180,E1 -12510.804,E2 -12510.804} C_VEL
LIN {X 0,Y 376.545,Z 489.673,A -85,B 0,C 180,E1 -12512.408,E2 -12512.408} C_VEL
LIN {X 0,Y 377.192,Z 482.091,A -85,B 0,C 180,E1 -12513.74,E2 -12513.74} C_VEL
LIN {X 0,Y 377.997,Z 472.883,A -85,B 0,C 180,E1 -12515.067,E2 -12515.067} C_VEL
LIN {X 0,Y 378.786,Z 462.65,A -85,B 0,C 180,E1 -12516.259,E2 -12516.259} C_VEL
LIN {X 0,Y 379.661,Z 451.287,A -85,B 0,C 180,E1 -12517.312,E2 -12517.312} C_VEL
LIN {X 0,Y 380.267,Z 439.481,A -85,B 0,C 180,E1 -12518.169,E2 -12518.169} C_VEL
LIN {X 0,Y 380.857,Z 427.094,A -85,B 0,C 180,E1 -12518.824,E2 -12518.824} C_VEL
LIN {X 0,Y 381.29,Z 413.277,A -85,B 0,C 180,E1 -12519.315,E2 -12519.315} C_VEL
LIN {X 0,Y 381.773,Z 383.473,A -85,B 0,C 180,E1 -12519.896,E2 -12519.896} C_VEL
LIN {X 0,Y 381.221,Z 377.656,A -85,B 0,C 180,E1 -12520.033,E2 -12520.033} C_VEL
LIN {X 0,Y 375.981,Z 358.928,A -85,B 0,C 180,E1 -12520.637,E2 -12520.637} C_VEL
LIN {X 0,Y 375.492,Z 353.111,A -85,B 0,C 180,E1 -12520.775,E2 -12520.775} C_VEL
LIN {X 0,Y 375.761,Z 328.574,A -85,B 0,C 180,E1 -12521.245,E2 -12521.245} C_VEL
LIN {X 0,Y 372.976,Z 314.492,A -85,B 0,C 180,E1 -12521.661,E2 -12521.661} C_VEL
LIN {X 0,Y 370.318,Z 305.874,A -85,B 0,C 180,E1 -12521.99,E2 -12521.99} C_VEL
LIN {X 0,Y 369.075,Z 299.509,A -85,B 0,C 180,E1 -12523.634,E2 -12523.634} C_VEL
LIN {X 0,Y 368.996,Z 299.517,A -85,B 0,C 180,E1 -12527.743,E2 -12527.743} C_VEL
LIN {X 0,Y 368.915,Z 299.53,A -85,B 0,C 180,E1 -12531.221,E2 -12531.221} C_VEL
LIN {X 0,Y 368.928,Z 299.532,A -85,B 0,C 180,E1 -12534.778,E2 -12534.778} C_VEL
LIN {X 0,Y 368.898,Z 299.534,A -85,B 0,C 180,E1 -12538.792,E2 -12538.792} C_VEL
LIN {X 0,Y 368.902,Z 299.529,A -85,B 0,C 180,E1 -12542.238,E2 -12542.238} C_VEL
LIN {X 0,Y 368.933,Z 299.531,A -85,B 0,C 180,E1 -12545.001,E2 -12545.001} C_VEL
LIN {X 0,Y 368.882,Z 299.533,A -85,B 0,C 180,E1 -12548.634,E2 -12548.634} C_VEL
LIN {X 0,Y 368.869,Z 299.533,A -85,B 0,C 180,E1 -12552.006,E2 -12552.006} C_VEL
LIN {X 0,Y 368.879,Z 299.537,A -85,B 0,C 180,E1 -12555.175,E2 -12555.175} C_VEL
LIN {X 0,Y 368.874,Z 299.533,A -85,B 0,C 180,E1 -12558.176,E2 -12558.176} C_VEL
LIN {X 0,Y 368.881,Z 299.538,A -85,B 0,C 180,E1 -12561.366,E2 -12561.366} C_VEL
LIN {X 0,Y 368.936,Z 299.527,A -85,B 0,C 180,E1 -12565.146,E2 -12565.146} C_VEL
LIN {X 0,Y 368.918,Z 299.528,A -85,B 0,C 180,E1 -12569.045,E2 -12569.045} C_VEL
LIN {X 0,Y 368.921,Z 299.532,A -85,B 0,C 180,E1 -12571.558,E2 -12571.558} C_VEL
LIN {X 0,Y 368.903,Z 299.53,A -85,B 0,C 180,E1 -12575.22,E2 -12575.22} C_VEL
LIN {X 0,Y 368.925,Z 299.531,A -85,B 0,C 180,E1 -12577.604,E2 -12577.604} C_VEL
LIN {X 0,Y 368.959,Z 299.522,A -85,B 0,C 180,E1 -12581.106,E2 -12581.106} C_VEL
LIN {X 0,Y 369.002,Z 299.518,A -85,B 0,C 180,E1 -12584.535,E2 -12584.535} C_VEL
LIN {X 0,Y 369.062,Z 299.509,A -85,B 0,C 180,E1 -12586.79,E2 -12586.79} C_VEL
LIN {X 0,Y 369.063,Z 299.515,A -85,B 0,C 180,E1 -12590.131,E2 -12590.131} C_VEL
LIN {X 0,Y 369.163,Z 299.497,A -85,B 0,C 180,E1 -12593.441,E2 -12593.441} C_VEL
LIN {X 0,Y 369.306,Z 299.481,A -85,B 0,C 180,E1 -12597.818,E2 -12597.818} C_VEL
LIN {X 0,Y 369.304,Z 299.484,A -85,B 0,C 180,E1 -12602.181,E2 -12602.181} C_VEL
LIN {X 0,Y 369.159,Z 299.502,A -85,B 0,C 180,E1 -12606.559,E2 -12606.559} C_VEL
LIN {X 0,Y 369.061,Z 299.51,A -85,B 0,C 180,E1 -12609.868,E2 -12609.868} C_VEL
LIN {X 0,Y 369.041,Z 299.512,A -85,B 0,C 180,E1 -12613.772,E2 -12613.772} C_VEL
LIN {X 0,Y 368.995,Z 299.517,A -85,B 0,C 180,E1 -12617.742,E2 -12617.742} C_VEL
LIN {X 0,Y 368.913,Z 299.529,A -85,B 0,C 180,E1 -12621.22,E2 -12621.22} C_VEL
LIN {X 0,Y 368.926,Z 299.532,A -85,B 0,C 180,E1 -12624.777,E2 -12624.777} C_VEL
LIN {X 0,Y 368.896,Z 299.535,A -85,B 0,C 180,E1 -12628.791,E2 -12628.791} C_VEL
LIN {X 0,Y 368.893,Z 299.53,A -85,B 0,C 180,E1 -12632.238,E2 -12632.238} C_VEL
LIN {X 0,Y 368.926,Z 299.532,A -85,B 0,C 180,E1 -12635,E2 -12635} C_VEL
LIN {X 0,Y 368.88,Z 299.533,A -85,B 0,C 180,E1 -12638.634,E2 -12638.634} C_VEL
LIN {X 0,Y 368.867,Z 299.533,A -85,B 0,C 180,E1 -12642.006,E2 -12642.006} C_VEL
LIN {X 0,Y 368.876,Z 299.538,A -85,B 0,C 180,E1 -12645.174,E2 -12645.174} C_VEL
LIN {X 0,Y 368.871,Z 299.533,A -85,B 0,C 180,E1 -12648.175,E2 -12648.175} C_VEL
LIN {X 0,Y 368.879,Z 299.538,A -85,B 0,C 180,E1 -12651.366,E2 -12651.366} C_VEL
LIN {X 0,Y 368.933,Z 299.528,A -85,B 0,C 180,E1 -12655.145,E2 -12655.145} C_VEL
LIN {X 0,Y 368.932,Z 299.528,A -85,B 0,C 180,E1 -12659.046,E2 -12659.046} C_VEL
LIN {X 0,Y 368.986,Z 299.713,A -85,B 0,C 180,E1 -12660.654,E2 -12660.654} C_VEL
LIN {X 0,Y 371.776,Z 313.788,A -85,B 0,C 180,E1 -12663.926,E2 -12663.926} C_VEL
LIN {X 0,Y 372.309,Z 317.26,A -85,B 0,C 180,E1 -12664.707,E2 -12664.707} C_VEL
LIN {X 0,Y 371.035,Z 333.601,A -85,B 0,C 180,E1 -12668.147,E2 -12668.147} C_VEL
LIN {X 0,Y 370.734,Z 337.958,A -85,B 0,C 180,E1 -12669.059,E2 -12669.059} C_VEL
LIN {X 0,Y 375.356,Z 373.135,A -85,B 0,C 180,E1 -12669.984,E2 -12669.984} C_VEL
LIN {X 0,Y 374.242,Z 447.203,A -85,B 0,C 180,E1 -12671.417,E2 -12671.417} C_VEL
LIN {X 0,Y 373.66,Z 460.374,A -85,B 0,C 180,E1 -12671.884,E2 -12671.884} C_VEL
LIN {X 0,Y 372.948,Z 472.513,A -85,B 0,C 180,E1 -12672.522,E2 -12672.522} C_VEL
LIN {X 0,Y 372.03,Z 484.756,A -85,B 0,C 180,E1 -12673.397,E2 -12673.397} C_VEL
LIN {X 0,Y 371.03,Z 496.375,A -85,B 0,C 180,E1 -12674.481,E2 -12674.481} C_VEL
LIN {X 0,Y 370.223,Z 506.856,A -85,B 0,C 180,E1 -12675.712,E2 -12675.712} C_VEL
LIN {X 0,Y 369.396,Z 516.249,A -85,B 0,C 180,E1 -12677.082,E2 -12677.082} C_VEL
LIN {X 0,Y 368.58,Z 525.341,A -85,B 0,C 180,E1 -12678.729,E2 -12678.729} C_VEL
LIN {X 0,Y 368.071,Z 532.667,A -85,B 0,C 180,E1 -12680.382,E2 -12680.382} C_VEL
LIN {X 0,Y 367.779,Z 537.609,A -85,B 0,C 180,E1 -12681.759,E2 -12681.759} C_VEL
LIN {X 0,Y 367.564,Z 542.404,A -85,B 0,C 180,E1 -12683.412,E2 -12683.412} C_VEL
LIN {X 0,Y 367.491,Z 546.065,A -85,B 0,C 180,E1 -12685.062,E2 -12685.062} C_VEL
LIN {X 0,Y 367.423,Z 548.694,A -85,B 0,C 180,E1 -12686.71,E2 -12686.71} C_VEL
LIN {X 0,Y 367.489,Z 549.933,A -85,B 0,C 180,E1 -12687.807,E2 -12687.807} C_VEL
LIN {X 0,Y 367.558,Z 550.744,A -85,B 0,C 180,E1 -12688.904,E2 -12688.904} C_VEL
LIN {X 0,Y 367.542,Z 551.127,A -85,B 0,C 180,E1 -12689.999,E2 -12689.999} C_VEL
LIN {X 0,Y 367.537,Z 551.121,A -85,B 0,C 180,E1 -12691.095,E2 -12691.095} C_VEL
LIN {X 0,Y 367.452,Z 550.726,A -85,B 0,C 180,E1 -12692.192,E2 -12692.192} C_VEL
LIN {X 0,Y 367.407,Z 549.928,A -85,B 0,C 180,E1 -12693.289,E2 -12693.289} C_VEL
LIN {X 0,Y 367.46,Z 548.697,A -85,B 0,C 180,E1 -12694.387,E2 -12694.387} C_VEL
LIN {X 0,Y 367.562,Z 545.014,A -85,B 0,C 180,E1 -12696.587,E2 -12696.587} C_VEL
LIN {X 0,Y 367.833,Z 541.052,A -85,B 0,C 180,E1 -12698.238,E2 -12698.238} C_VEL
LIN {X 0,Y 368.246,Z 535.97,A -85,B 0,C 180,E1 -12699.89,E2 -12699.89} C_VEL
LIN {X 0,Y 368.914,Z 529.608,A -85,B 0,C 180,E1 -12701.538,E2 -12701.538} C_VEL
LIN {X 0,Y 369.961,Z 521.673,A -85,B 0,C 180,E1 -12703.176,E2 -12703.176} C_VEL
LIN {X 0,Y 370.863,Z 513.622,A -85,B 0,C 180,E1 -12704.54,E2 -12704.54} C_VEL
LIN {X 0,Y 372.007,Z 503.81,A -85,B 0,C 180,E1 -12705.898,E2 -12705.898} C_VEL
LIN {X 0,Y 373.267,Z 492.893,A -85,B 0,C 180,E1 -12707.108,E2 -12707.108} C_VEL
LIN {X 0,Y 374.408,Z 482.219,A -85,B 0,C 180,E1 -12708.042,E2 -12708.042} C_VEL
LIN {X 0,Y 375.572,Z 469.391,A -85,B 0,C 180,E1 -12708.902,E2 -12708.902} C_VEL
LIN {X 0,Y 376.506,Z 456.385,A -85,B 0,C 180,E1 -12709.526,E2 -12709.526} C_VEL
LIN {X 0,Y 377.105,Z 443.898,A -85,B 0,C 180,E1 -12709.909,E2 -12709.909} C_VEL
LIN {X 0,Y 378.312,Z 372.669,A -85,B 0,C 180,E1 -12711.292,E2 -12711.292} C_VEL
LIN {X 0,Y 374.79,Z 350.976,A -85,B 0,C 180,E1 -12711.98,E2 -12711.98} C_VEL
LIN {X 0,Y 372.121,Z 337.443,A -85,B 0,C 180,E1 -12712.456,E2 -12712.456} C_VEL
LIN {X 0,Y 373.55,Z 322.659,A -85,B 0,C 180,E1 -12715.64,E2 -12715.64} C_VEL
LIN {X 0,Y 373.189,Z 318.659,A -85,B 0,C 180,E1 -12716.568,E2 -12716.568} C_VEL
LIN {X 0,Y 370.836,Z 307.455,A -85,B 0,C 180,E1 -12719.334,E2 -12719.334} C_VEL
LIN {X 0,Y 368.917,Z 299.534,A -85,B 0,C 180,E1 -12721.432,E2 -12721.432} C_VEL
LIN {X 0,Y 368.926,Z 299.534,A -85,B 0,C 180,E1 -12725.001,E2 -12725.001} C_VEL
LIN {X 0,Y 368.903,Z 299.533,A -85,B 0,C 180,E1 -12728.639,E2 -12728.639} C_VEL
LIN {X 0,Y 368.878,Z 299.534,A -85,B 0,C 180,E1 -12732.009,E2 -12732.009} C_VEL
LIN {X 0,Y 368.877,Z 299.535,A -85,B 0,C 180,E1 -12735.175,E2 -12735.175} C_VEL
LIN {X 0,Y 368.88,Z 299.537,A -85,B 0,C 180,E1 -12738.177,E2 -12738.177} C_VEL
LIN {X 0,Y 368.906,Z 299.528,A -85,B 0,C 180,E1 -12741.359,E2 -12741.359} C_VEL
LIN {X 0,Y 368.933,Z 299.523,A -85,B 0,C 180,E1 -12745.146,E2 -12745.146} C_VEL
LIN {X 0,Y 368.925,Z 299.527,A -85,B 0,C 180,E1 -12749.046,E2 -12749.046} C_VEL
LIN {X 0,Y 368.959,Z 299.523,A -85,B 0,C 180,E1 -12752.796,E2 -12752.796} C_VEL
LIN {X 0,Y 368.941,Z 299.52,A -85,B 0,C 180,E1 -12756.113,E2 -12756.113} C_VEL
LIN {X 0,Y 368.933,Z 299.519,A -85,B 0,C 180,E1 -12759.947,E2 -12759.947} C_VEL
LIN {X 0,Y 368.972,Z 299.516,A -85,B 0,C 180,E1 -12763.399,E2 -12763.399} C_VEL
LIN {X 0,Y 369.054,Z 299.512,A -85,B 0,C 180,E1 -12766.79,E2 -12766.79} C_VEL
LIN {X 0,Y 369.064,Z 299.511,A -85,B 0,C 180,E1 -12770.132,E2 -12770.132} C_VEL
LIN {X 0,Y 369.184,Z 299.491,A -85,B 0,C 180,E1 -12772.342,E2 -12772.342} C_VEL
LIN {X 0,Y 369.141,Z 299.503,A -85,B 0,C 180,E1 -12774.538,E2 -12774.538} C_VEL
LIN {X 0,Y 369.316,Z 299.478,A -85,B 0,C 180,E1 -12777.819,E2 -12777.819} C_VEL
LIN {X 0,Y 369.455,Z 299.458,A -85,B 0,C 180,E1 -12780,E2 -12780} C_VEL
LIN {X 0,Y 369.315,Z 299.477,A -85,B 0,C 180,E1 -12782.181,E2 -12782.181} C_VEL
LIN {X 0,Y 369.201,Z 299.492,A -85,B 0,C 180,E1 -12786.616,E2 -12786.616} C_VEL
LIN {X 0,Y 369.134,Z 299.5,A -85,B 0,C 180,E1 -12788.761,E2 -12788.761} C_VEL
LIN {X 0,Y 369.002,Z 299.516,A -85,B 0,C 180,E1 -12792.094,E2 -12792.094} C_VEL
LIN {X 0,Y 368.995,Z 299.521,A -85,B 0,C 180,E1 -12795.465,E2 -12795.465} C_VEL
LIN {X 0,Y 368.955,Z 299.525,A -85,B 0,C 180,E1 -12798.895,E2 -12798.895} C_VEL
LIN {X 0,Y 368.929,Z 299.525,A -85,B 0,C 180,E1 -12802.396,E2 -12802.396} C_VEL
LIN {X 0,Y 368.998,Z 299.518,A -85,B 0,C 180,E1 -12805.981,E2 -12805.981} C_VEL
LIN {X 0,Y 368.913,Z 299.53,A -85,B 0,C 180,E1 -12809.691,E2 -12809.691} C_VEL
LIN {X 0,Y 368.895,Z 299.529,A -85,B 0,C 180,E1 -12813.044,E2 -12813.044} C_VEL
LIN {X 0,Y 368.915,Z 299.527,A -85,B 0,C 180,E1 -12816.198,E2 -12816.198} C_VEL
LIN {X 0,Y 368.876,Z 299.531,A -85,B 0,C 180,E1 -12818.957,E2 -12818.957} C_VEL
LIN {X 0,Y 368.871,Z 299.536,A -85,B 0,C 180,E1 -12822.009,E2 -12822.009} C_VEL
LIN {X 0,Y 368.877,Z 299.537,A -85,B 0,C 180,E1 -12825.176,E2 -12825.176} C_VEL
LIN {X 0,Y 368.868,Z 299.537,A -85,B 0,C 180,E1 -12828.177,E2 -12828.177} C_VEL
LIN {X 0,Y 368.876,Z 299.537,A -85,B 0,C 180,E1 -12831.367,E2 -12831.367} C_VEL
LIN {X 0,Y 368.937,Z 299.524,A -85,B 0,C 180,E1 -12835.147,E2 -12835.147} C_VEL
LIN {X 0,Y 368.975,Z 299.612,A -85,B 0,C 180,E1 -12836.616,E2 -12836.616} C_VEL
LIN {X 0,Y 370.549,Z 306.634,A -85,B 0,C 180,E1 -12838.469,E2 -12838.469} C_VEL
LIN {X 0,Y 377.18,Z 322.537,A -85,B 0,C 180,E1 -12839.286,E2 -12839.286} C_VEL
LIN {X 0,Y 379.048,Z 330.571,A -85,B 0,C 180,E1 -12839.582,E2 -12839.582} C_VEL
LIN {X 0,Y 377.408,Z 414.049,A -85,B 0,C 180,E1 -12841.207,E2 -12841.207} C_VEL
LIN {X 0,Y 376.934,Z 427.393,A -85,B 0,C 180,E1 -12841.694,E2 -12841.694} C_VEL
LIN {X 0,Y 376.1,Z 440.176,A -85,B 0,C 180,E1 -12842.377,E2 -12842.377} C_VEL
LIN {X 0,Y 375.119,Z 452.359,A -85,B 0,C 180,E1 -12843.28,E2 -12843.28} C_VEL
LIN {X 0,Y 374.073,Z 463.973,A -85,B 0,C 180,E1 -12844.399,E2 -12844.399} C_VEL
LIN {X 0,Y 372.854,Z 474.334,A -85,B 0,C 180,E1 -12845.65,E2 -12845.65} C_VEL
LIN {X 0,Y 371.653,Z 484.429,A -85,B 0,C 180,E1 -12847.192,E2 -12847.192} C_VEL
LIN {X 0,Y 370.493,Z 493.239,A -85,B 0,C 180,E1 -12848.875,E2 -12848.875} C_VEL
LIN {X 0,Y 369.57,Z 500.208,A -85,B 0,C 180,E1 -12850.562,E2 -12850.562} C_VEL
LIN {X 0,Y 368.861,Z 505.89,A -85,B 0,C 180,E1 -12852.302,E2 -12852.302} C_VEL
LIN {X 0,Y 368.321,Z 510.049,A -85,B 0,C 180,E1 -12853.939,E2 -12853.939} C_VEL
LIN {X 0,Y 367.902,Z 513.246,A -85,B 0,C 180,E1 -12855.622,E2 -12855.622} C_VEL
LIN {X 0,Y 367.743,Z 515.206,A -85,B 0,C 180,E1 -12857.08,E2 -12857.08} C_VEL
LIN {X 0,Y 367.477,Z 516.674,A -85,B 0,C 180,E1 -12858.975,E2 -12858.975} C_VEL
LIN {X 0,Y 367.415,Z 516.917,A -85,B 0,C 180,E1 -12861.198,E2 -12861.198} C_VEL
LIN {X 0,Y 367.481,Z 516.432,A -85,B 0,C 180,E1 -12862.307,E2 -12862.307} C_VEL
LIN {X 0,Y 367.606,Z 515.12,A -85,B 0,C 180,E1 -12863.807,E2 -12863.807} C_VEL
LIN {X 0,Y 367.713,Z 511.505,A -85,B 0,C 180,E1 -12866.165,E2 -12866.165} C_VEL
LIN {X 0,Y 368.029,Z 507.76,A -85,B 0,C 180,E1 -12867.812,E2 -12867.812} C_VEL
LIN {X 0,Y 368.321,Z 502.919,A -85,B 0,C 180,E1 -12869.454,E2 -12869.454} C_VEL
LIN {X 0,Y 368.933,Z 496.808,A -85,B 0,C 180,E1 -12871.092,E2 -12871.092} C_VEL
LIN {X 0,Y 369.608,Z 489.227,A -85,B 0,C 180,E1 -12872.725,E2 -12872.725} C_VEL
LIN {X 0,Y 370.446,Z 479.707,A -85,B 0,C 180,E1 -12874.353,E2 -12874.353} C_VEL
LIN {X 0,Y 371.306,Z 469.893,A -85,B 0,C 180,E1 -12875.704,E2 -12875.704} C_VEL
LIN {X 0,Y 372.219,Z 458.846,A -85,B 0,C 180,E1 -12876.914,E2 -12876.914} C_VEL
LIN {X 0,Y 373.112,Z 446.292,A -85,B 0,C 180,E1 -12877.986,E2 -12877.986} C_VEL
LIN {X 0,Y 373.698,Z 433.803,A -85,B 0,C 180,E1 -12878.79,E2 -12878.79} C_VEL
LIN {X 0,Y 374.285,Z 420.38,A -85,B 0,C 180,E1 -12879.389,E2 -12879.389} C_VEL
LIN {X 0,Y 374.655,Z 407.15,A -85,B 0,C 180,E1 -12879.751,E2 -12879.751} C_VEL
LIN {X 0,Y 375.492,Z 353.111,A -85,B 0,C 180,E1 -12880.775,E2 -12880.775} C_VEL
LIN {X 0,Y 375.025,Z 347.286,A -85,B 0,C 180,E1 -12880.912,E2 -12880.912} C_VEL
LIN {X 0,Y 372.378,Z 337.945,A -85,B 0,C 180,E1 -12881.224,E2 -12881.224} C_VEL
LIN {X 0,Y 368.649,Z 326.786,A -85,B 0,C 180,E1 -12881.633,E2 -12881.633} C_VEL
LIN {X 0,Y 367.848,Z 322.933,A -85,B 0,C 180,E1 -12881.751,E2 -12881.751} C_VEL
LIN {X 0,Y 365.935,Z 314.944,A -85,B 0,C 180,E1 -12882.011,E2 -12882.011} C_VEL
LIN {X 0,Y 363.18,Z 306.181,A -85,B 0,C 180,E1 -12882.362,E2 -12882.362} C_VEL
LIN {X 0,Y 361.995,Z 300.391,A -85,B 0,C 180,E1 -12883.894,E2 -12883.894} C_VEL
LIN {X 0,Y 361.934,Z 300.401,A -85,B 0,C 180,E1 -12886.935,E2 -12886.935} C_VEL
LIN {X 0,Y 361.892,Z 300.405,A -85,B 0,C 180,E1 -12890.461,E2 -12890.461} C_VEL
LIN {X 0,Y 361.899,Z 300.402,A -85,B 0,C 180,E1 -12894.113,E2 -12894.113} C_VEL
LIN {X 0,Y 361.84,Z 300.409,A -85,B 0,C 180,E1 -12897.785,E2 -12897.785} C_VEL
LIN {X 0,Y 361.852,Z 300.411,A -85,B 0,C 180,E1 -12901.285,E2 -12901.285} C_VEL
LIN {X 0,Y 361.859,Z 300.407,A -85,B 0,C 180,E1 -12904.281,E2 -12904.281} C_VEL
LIN {X 0,Y 361.865,Z 300.411,A -85,B 0,C 180,E1 -12907.222,E2 -12907.222} C_VEL
LIN {X 0,Y 361.816,Z 300.414,A -85,B 0,C 180,E1 -12910.751,E2 -12910.751} C_VEL
LIN {X 0,Y 361.817,Z 300.411,A -85,B 0,C 180,E1 -12914.37,E2 -12914.37} C_VEL
LIN {X 0,Y 361.834,Z 300.414,A -85,B 0,C 180,E1 -12917.569,E2 -12917.569} C_VEL
LIN {X 0,Y 361.847,Z 300.413,A -85,B 0,C 180,E1 -12921.572,E2 -12921.572} C_VEL
LIN {X 0,Y 361.875,Z 300.404,A -85,B 0,C 180,E1 -12924.656,E2 -12924.656} C_VEL
LIN {X 0,Y 361.842,Z 300.409,A -85,B 0,C 180,E1 -12928.37,E2 -12928.37} C_VEL
LIN {X 0,Y 361.871,Z 300.405,A -85,B 0,C 180,E1 -12930.952,E2 -12930.952} C_VEL
LIN {X 0,Y 361.873,Z 300.404,A -85,B 0,C 180,E1 -12934.705,E2 -12934.705} C_VEL
LIN {X 0,Y 361.866,Z 300.407,A -85,B 0,C 180,E1 -12938.345,E2 -12938.345} C_VEL
LIN {X 0,Y 361.926,Z 300.403,A -85,B 0,C 180,E1 -12942.084,E2 -12942.084} C_VEL
LIN {X 0,Y 361.967,Z 300.394,A -85,B 0,C 180,E1 -12945.379,E2 -12945.379} C_VEL
LIN {X 0,Y 361.969,Z 300.393,A -85,B 0,C 180,E1 -12948.804,E2 -12948.804} C_VEL
LIN {X 0,Y 362.082,Z 300.385,A -85,B 0,C 180,E1 -12952.191,E2 -12952.191} C_VEL
LIN {X 0,Y 362.096,Z 300.381,A -85,B 0,C 180,E1 -12954.431,E2 -12954.431} C_VEL
LIN {X 0,Y 362.268,Z 300.357,A -85,B 0,C 180,E1 -12957.776,E2 -12957.776} C_VEL
LIN {X 0,Y 362.198,Z 300.364,A -85,B 0,C 180,E1 -12961.112,E2 -12961.112} C_VEL
LIN {X 0,Y 362.267,Z 300.361,A -85,B 0,C 180,E1 -12962.223,E2 -12962.223} C_VEL
LIN {X 0,Y 362.123,Z 300.377,A -85,B 0,C 180,E1 -12966.687,E2 -12966.687} C_VEL
LIN {X 0,Y 361.998,Z 300.391,A -85,B 0,C 180,E1 -12970.063,E2 -12970.063} C_VEL
LIN {X 0,Y 362.002,Z 300.389,A -85,B 0,C 180,E1 -12973.898,E2 -12973.898} C_VEL
LIN {X 0,Y 361.931,Z 300.401,A -85,B 0,C 180,E1 -12976.934,E2 -12976.934} C_VEL
